LIN {X 0,Y 340.456,Z 505.145,A -85,B 0,C 180,E1 -14305.856,E2 -14305.856} C_VEL
LIN {X 0,Y 340.517,Z 502.884,A -85,B 0,C 180,E1 -14307.19,E2 -14307.19} C_VEL
LIN {X 0,Y 341.184,Z 502.798,A -85,B 0,C 180,E1 -14309.999,E2 -14309.999} C_VEL
LIN {X 0,Y 341.171,Z 502.802,A -85,B 0,C 180,E1 -14312.361,E2 -14312.361} C_VEL
LIN {X 0,Y 341.077,Z 502.809,A -85,B 0,C 180,E1 -14317.101,E2 -14317.101} C_VEL
LIN {X 0,Y 340.872,Z 502.837,A -85,B 0,C 180,E1 -14320.693,E2 -14320.693} C_VEL
LIN {X 0,Y 340.863,Z 502.841,A -85,B 0,C 180,E1 -14324.324,E2 -14324.324} C_VEL
LIN {X 0,Y 340.838,Z 502.842,A -85,B 0,C 180,E1 -14328.466,E2 -14328.466} C_VEL
LIN {X 0,Y 340.754,Z 502.851,A -85,B 0,C 180,E1 -14331.856,E2 -14331.856} C_VEL
LIN {X 0,Y 340.773,Z 502.848,A -85,B 0,C 180,E1 -14335.664,E2 -14335.664} C_VEL
LIN {X 0,Y 340.742,Z 502.855,A -85,B 0,C 180,E1 -14338.319,E2 -14338.319} C_VEL
LIN {X 0,Y 340.704,Z 502.855,A -85,B 0,C 180,E1 -14341.043,E2 -14341.043} C_VEL
LIN {X 0,Y 340.717,Z 502.854,A -85,B 0,C 180,E1 -14345.278,E2 -14345.278} C_VEL
LIN {X 0,Y 340.709,Z 502.858,A -85,B 0,C 180,E1 -14348.386,E2 -14348.386} C_VEL
LIN {X 0,Y 340.719,Z 502.859,A -85,B 0,C 180,E1 -14352.049,E2 -14352.049} C_VEL
LIN {X 0,Y 340.721,Z 502.854,A -85,B 0,C 180,E1 -14355.467,E2 -14355.467} C_VEL
LIN {X 0,Y 340.722,Z 502.853,A -85,B 0,C 180,E1 -14358.81,E2 -14358.81} C_VEL
LIN {X 0,Y 340.063,Z 502.939,A -85,B 0,C 180,E1 -14359.797,E2 -14359.797} C_VEL
LIN {X 0,Y 337.229,Z 503.295,A -85,B 0,C 180,E1 -14361.402,E2 -14361.402} C_VEL
LIN {X 0,Y 334.812,Z 503.598,A -85,B 0,C 180,E1 -14362.702,E2 -14362.702} C_VEL
LIN {X 0,Y 333.759,Z 503.725,A -85,B 0,C 180,E1 -14363.708,E2 -14363.708} C_VEL
LIN {X 0,Y 333.664,Z 503.734,A -85,B 0,C 180,E1 -14364.048,E2 -14364.048} C_VEL
LIN {X 0,Y 333.641,Z 503.736,A -85,B 0,C 180,E1 -14367.413,E2 -14367.413} C_VEL
LIN {X 0,Y 333.708,Z 503.726,A -85,B 0,C 180,E1 -14371.028,E2 -14371.028} C_VEL
LIN {X 0,Y 333.733,Z 503.727,A -85,B 0,C 180,E1 -14373.753,E2 -14373.753} C_VEL
LIN {X 0,Y 333.717,Z 503.731,A -85,B 0,C 180,E1 -14377.914,E2 -14377.914} C_VEL
LIN {X 0,Y 333.792,Z 503.719,A -85,B 0,C 180,E1 -14381.589,E2 -14381.589} C_VEL
LIN {X 0,Y 333.805,Z 503.717,A -85,B 0,C 180,E1 -14385.576,E2 -14385.576} C_VEL
LIN {X 0,Y 333.835,Z 503.711,A -85,B 0,C 180,E1 -14389.078,E2 -14389.078} C_VEL
LIN {X 0,Y 334.023,Z 503.687,A -85,B 0,C 180,E1 -14392.747,E2 -14392.747} C_VEL
LIN {X 0,Y 333.81,Z 503.714,A -85,B 0,C 180,E1 -14395.169,E2 -14395.169} C_VEL
LIN {X 0,Y 334.105,Z 503.681,A -85,B 0,C 180,E1 -14397.589,E2 -14397.589} C_VEL
LIN {X 0,Y 334.245,Z 503.663,A -85,B 0,C 180,E1 -14400,E2 -14400} C_VEL
LIN {X 0,Y 334.106,Z 503.678,A -85,B 0,C 180,E1 -14402.411,E2 -14402.411} C_VEL
LIN {X 0,Y 334.023,Z 503.689,A -85,B 0,C 180,E1 -14407.252,E2 -14407.252} C_VEL
LIN {X 0,Y 333.832,Z 503.711,A -85,B 0,C 180,E1 -14410.922,E2 -14410.922} C_VEL
LIN {X 0,Y 333.805,Z 503.714,A -85,B 0,C 180,E1 -14414.634,E2 -14414.634} C_VEL
LIN {X 0,Y 333.793,Z 503.716,A -85,B 0,C 180,E1 -14418.655,E2 -14418.655} C_VEL
LIN {X 0,Y 333.689,Z 503.73,A -85,B 0,C 180,E1 -14422.278,E2 -14422.278} C_VEL
LIN {X 0,Y 333.733,Z 503.724,A -85,B 0,C 180,E1 -14426.246,E2 -14426.246} C_VEL
LIN {X 0,Y 333.709,Z 503.727,A -85,B 0,C 180,E1 -14428.972,E2 -14428.972} C_VEL
LIN {X 0,Y 333.648,Z 503.734,A -85,B 0,C 180,E1 -14432.589,E2 -14432.589} C_VEL
LIN {X 0,Y 333.674,Z 503.732,A -85,B 0,C 180,E1 -14436.139,E2 -14436.139} C_VEL
LIN {X 0,Y 333.644,Z 503.737,A -85,B 0,C 180,E1 -14439.193,E2 -14439.193} C_VEL
LIN {X 0,Y 333.63,Z 503.736,A -85,B 0,C 180,E1 -14442.5,E2 -14442.5} C_VEL
LIN {X 0,Y 333.645,Z 503.736,A -85,B 0,C 180,E1 -14445.964,E2 -14445.964} C_VEL
LIN {X 0,Y 333.654,Z 503.738,A -85,B 0,C 180,E1 -14449.314,E2 -14449.314} C_VEL
LIN {X 0,Y 333.787,Z 503.868,A -85,B 0,C 180,E1 -14452.482,E2 -14452.482} C_VEL
LIN {X 0,Y 334.922,Z 510.332,A -85,B 0,C 180,E1 -14456.216,E2 -14456.216} C_VEL
LIN {X 0,Y 335.329,Z 513.013,A -85,B 0,C 180,E1 -14457.717,E2 -14457.717} C_VEL
LIN {X 0,Y 334.834,Z 518.114,A -85,B 0,C 180,E1 -14460.446,E2 -14460.446} C_VEL
LIN {X 0,Y 333.958,Z 525.622,A -85,B 0,C 180,E1 -14464.379,E2 -14464.379} C_VEL
LIN {X 0,Y 333.231,Z 532.887,A -85,B 0,C 180,E1 -14468.122,E2 -14468.122} C_VEL
LIN {X 0,Y 332.697,Z 540.288,A -85,B 0,C 180,E1 -14471.914,E2 -14471.914} C_VEL
LIN {X 0,Y 332.542,Z 543.414,A -85,B 0,C 180,E1 -14473.502,E2 -14473.502} C_VEL
LIN {X 0,Y 333.88,Z 554.918,A -85,B 0,C 180,E1 -14474.002,E2 -14474.002} C_VEL
LIN {X 0,Y 334.682,Z 563.382,A -85,B 0,C 180,E1 -14474.509,E2 -14474.509} C_VEL
LIN {X 0,Y 335.194,Z 571.374,A -85,B 0,C 180,E1 -14475.115,E2 -14475.115} C_VEL
LIN {X 0,Y 335.488,Z 578.299,A -85,B 0,C 180,E1 -14475.751,E2 -14475.751} C_VEL
LIN {X 0,Y 334.937,Z 586.572,A -85,B 0,C 180,E1 -14476.656,E2 -14476.656} C_VEL
LIN {X 0,Y 334.225,Z 594.387,A -85,B 0,C 180,E1 -14477.708,E2 -14477.708} C_VEL
LIN {X 0,Y 333.675,Z 600.834,A -85,B 0,C 180,E1 -14478.766,E2 -14478.766} C_VEL
LIN {X 0,Y 333.106,Z 606.952,A -85,B 0,C 180,E1 -14479.977,E2 -14479.977} C_VEL
LIN {X 0,Y 332.646,Z 613.19,A -85,B 0,C 180,E1 -14481.496,E2 -14481.496} C_VEL
LIN {X 0,Y 332.216,Z 618.901,A -85,B 0,C 180,E1 -14483.319,E2 -14483.319} C_VEL
LIN {X 0,Y 332.065,Z 621.825,A -85,B 0,C 180,E1 -14484.512,E2 -14484.512} C_VEL
LIN {X 0,Y 332.055,Z 625.07,A -85,B 0,C 180,E1 -14486.36,E2 -14486.36} C_VEL
LIN {X 0,Y 331.969,Z 626.568,A -85,B 0,C 180,E1 -14487.574,E2 -14487.574} C_VEL
LIN {X 0,Y 331.973,Z 627.512,A -85,B 0,C 180,E1 -14488.788,E2 -14488.788} C_VEL
LIN {X 0,Y 332.038,Z 627.871,A -85,B 0,C 180,E1 -14490.001,E2 -14490.001} C_VEL
LIN {X 0,Y 331.97,Z 627.733,A -85,B 0,C 180,E1 -14491.214,E2 -14491.214} C_VEL
LIN {X 0,Y 331.964,Z 627.113,A -85,B 0,C 180,E1 -14492.427,E2 -14492.427} C_VEL
LIN {X 0,Y 332.051,Z 626.001,A -85,B 0,C 180,E1 -14493.641,E2 -14493.641} C_VEL
LIN {X 0,Y 332.1,Z 624.338,A -85,B 0,C 180,E1 -14494.856,E2 -14494.856} C_VEL
LIN {X 0,Y 332.553,Z 618.216,A -85,B 0,C 180,E1 -14497.896,E2 -14497.896} C_VEL
LIN {X 0,Y 333.215,Z 613.214,A -85,B 0,C 180,E1 -14499.715,E2 -14499.715} C_VEL
LIN {X 0,Y 334.003,Z 607.935,A -85,B 0,C 180,E1 -14501.224,E2 -14501.224} C_VEL
LIN {X 0,Y 335.091,Z 601.437,A -85,B 0,C 180,E1 -14502.723,E2 -14502.723} C_VEL
LIN {X 0,Y 336.316,Z 593.514,A -85,B 0,C 180,E1 -14504.214,E2 -14504.214} C_VEL
LIN {X 0,Y 337.945,Z 583.56,A -85,B 0,C 180,E1 -14505.686,E2 -14505.686} C_VEL
LIN {X 0,Y 338.393,Z 575.402,A -85,B 0,C 180,E1 -14506.733,E2 -14506.733} C_VEL
LIN {X 0,Y 338.314,Z 568.475,A -85,B 0,C 180,E1 -14507.531,E2 -14507.531} C_VEL
LIN {X 0,Y 337.193,Z 558.94,A -85,B 0,C 180,E1 -14508.552,E2 -14508.552} C_VEL
LIN {X 0,Y 335.395,Z 550.189,A -85,B 0,C 180,E1 -14509.448,E2 -14509.448} C_VEL
LIN {X 0,Y 333.241,Z 542.09,A -85,B 0,C 180,E1 -14510.224,E2 -14510.224} C_VEL
LIN {X 0,Y 333.215,Z 541.572,A -85,B 0,C 180,E1 -14510.366,E2 -14510.366} C_VEL
LIN {X 0,Y 333.935,Z 535.173,A -85,B 0,C 180,E1 -14514.23,E2 -14514.23} C_VEL
LIN {X 0,Y 334.748,Z 530.134,A -85,B 0,C 180,E1 -14517.51,E2 -14517.51} C_VEL
LIN {X 0,Y 335.654,Z 525.473,A -85,B 0,C 180,E1 -14520.855,E2 -14520.855} C_VEL
LIN {X 0,Y 336.223,Z 522.467,A -85,B 0,C 180,E1 -14523.268,E2 -14523.268} C_VEL
LIN {X 0,Y 336.353,Z 519.746,A -85,B 0,C 180,E1 -14525.807,E2 -14525.807} C_VEL
LIN {X 0,Y 336.02,Z 517.109,A -85,B 0,C 180,E1 -14528.864,E2 -14528.864} C_VEL
LIN {X 0,Y 335.687,Z 514.987,A -85,B 0,C 180,E1 -14532.065,E2 -14532.065} C_VEL
LIN {X 0,Y 335.387,Z 513.454,A -85,B 0,C 180,E1 -14535.437,E2 -14535.437} C_VEL
LIN {X 0,Y 335.245,Z 512.57,A -85,B 0,C 180,E1 -14539,E2 -14539} C_VEL
LIN {X 0,Y 335.145,Z 512.414,A -85,B 0,C 180,E1 -14542.546,E2 -14542.546} C_VEL
LIN {X 0,Y 335.113,Z 512.774,A -85,B 0,C 180,E1 -14545.511,E2 -14545.511} C_VEL
LIN {X 0,Y 334.894,Z 513.56,A -85,B 0,C 180,E1 -14548.356,E2 -14548.356} C_VEL
LIN {X 0,Y 334.407,Z 515.069,A -85,B 0,C 180,E1 -14551.969,E2 -14551.969} C_VEL
LIN {X 0,Y 333.979,Z 516.753,A -85,B 0,C 180,E1 -14555.111,E2 -14555.111} C_VEL
LIN {X 0,Y 333.557,Z 519.216,A -85,B 0,C 180,E1 -14559.011,E2 -14559.011} C_VEL
LIN {X 0,Y 333.507,Z 520.041,A -85,B 0,C 180,E1 -14559.935,E2 -14559.935} C_VEL
LIN {X 0,Y 337.947,Z 531.73,A -85,B 0,C 180,E1 -14561.371,E2 -14561.371} C_VEL
LIN {X 0,Y 340.475,Z 541.669,A -85,B 0,C 180,E1 -14562.641,E2 -14562.641} C_VEL
LIN {X 0,Y 341.129,Z 546.298,A -85,B 0,C 180,E1 -14563.236,E2 -14563.236} C_VEL
LIN {X 0,Y 339.871,Z 554.77,A -85,B 0,C 180,E1 -14564.252,E2 -14564.252} C_VEL
LIN {X 0,Y 338.492,Z 563.651,A -85,B 0,C 180,E1 -14565.573,E2 -14565.573} C_VEL
LIN {X 0,Y 337.09,Z 571.617,A -85,B 0,C 180,E1 -14567.049,E2 -14567.049} C_VEL
LIN {X 0,Y 335.873,Z 577.991,A -85,B 0,C 180,E1 -14568.534,E2 -14568.534} C_VEL
LIN {X 0,Y 335.057,Z 582.231,A -85,B 0,C 180,E1 -14569.73,E2 -14569.73} C_VEL
LIN {X 0,Y 334.387,Z 586.055,A -85,B 0,C 180,E1 -14571.053,E2 -14571.053} C_VEL
LIN {X 0,Y 333.402,Z 589.807,A -85,B 0,C 180,E1 -14572.734,E2 -14572.734} C_VEL
LIN {X 0,Y 333.118,Z 591.829,A -85,B 0,C 180,E1 -14573.945,E2 -14573.945} C_VEL
LIN {X 0,Y 332.982,Z 593.306,A -85,B 0,C 180,E1 -14575.157,E2 -14575.157} C_VEL
LIN {X 0,Y 332.648,Z 594.219,A -85,B 0,C 180,E1 -14576.366,E2 -14576.366} C_VEL
LIN {X 0,Y 332.405,Z 594.638,A -85,B 0,C 180,E1 -14577.577,E2 -14577.577} C_VEL
LIN {X 0,Y 332.209,Z 594.58,A -85,B 0,C 180,E1 -14578.788,E2 -14578.788} C_VEL
LIN {X 0,Y 332.136,Z 594.037,A -85,B 0,C 180,E1 -14580,E2 -14580} C_VEL
LIN {X 0,Y 332.096,Z 592.929,A -85,B 0,C 180,E1 -14581.213,E2 -14581.213} C_VEL
LIN {X 0,Y 332.155,Z 590.254,A -85,B 0,C 180,E1 -14583.032,E2 -14583.032} C_VEL
LIN {X 0,Y 332.366,Z 586.242,A -85,B 0,C 180,E1 -14584.852,E2 -14584.852} C_VEL
LIN {X 0,Y 332.593,Z 580.732,A -85,B 0,C 180,E1 -14586.703,E2 -14586.703} C_VEL
LIN {X 0,Y 332.978,Z 575.054,A -85,B 0,C 180,E1 -14588.191,E2 -14588.191} C_VEL
LIN {X 0,Y 333.406,Z 567.758,A -85,B 0,C 180,E1 -14589.709,E2 -14589.709} C_VEL
LIN {X 0,Y 334.005,Z 559.596,A -85,B 0,C 180,E1 -14591.07,E2 -14591.07} C_VEL
LIN {X 0,Y 334.497,Z 551.909,A -85,B 0,C 180,E1 -14592.129,E2 -14592.129} C_VEL
LIN {X 0,Y 335.116,Z 542.576,A -85,B 0,C 180,E1 -14593.184,E2 -14593.184} C_VEL
LIN {X 0,Y 335.377,Z 535.383,A -85,B 0,C 180,E1 -14593.844,E2 -14593.844} C_VEL
LIN {X 0,Y 333.631,Z 524.142,A -85,B 0,C 180,E1 -14594.72,E2 -14594.72} C_VEL
LIN {X 0,Y 332.344,Z 514.848,A -85,B 0,C 180,E1 -14595.288,E2 -14595.288} C_VEL
LIN {X 0,Y 332.367,Z 511.054,A -85,B 0,C 180,E1 -14598.493,E2 -14598.493} C_VEL
LIN {X 0,Y 332.502,Z 506.577,A -85,B 0,C 180,E1 -14602.362,E2 -14602.362} C_VEL
LIN {X 0,Y 332.729,Z 503.94,A -85,B 0,C 180,E1 -14604.792,E2 -14604.792} C_VEL
LIN {X 0,Y 333.7,Z 507.775,A -85,B 0,C 180,E1 -14606.924,E2 -14606.924} C_VEL
LIN {X 0,Y 333.738,Z 511.614,A -85,B 0,C 180,E1 -14608.97,E2 -14608.97} C_VEL
LIN {X 0,Y 333.445,Z 518.337,A -85,B 0,C 180,E1 -14612.533,E2 -14612.533} C_VEL
LIN {X 0,Y 333.168,Z 525.241,A -85,B 0,C 180,E1 -14616.203,E2 -14616.203} C_VEL
LIN {X 0,Y 332.985,Z 529.458,A -85,B 0,C 180,E1 -14618.447,E2 -14618.447} C_VEL
LIN {X 0,Y 335.211,Z 539.502,A -85,B 0,C 180,E1 -14619.054,E2 -14619.054} C_VEL
LIN {X 0,Y 336.797,Z 548.312,A -85,B 0,C 180,E1 -14619.721,E2 -14619.721} C_VEL
LIN {X 0,Y 337.709,Z 557.401,A -85,B 0,C 180,E1 -14620.536,E2 -14620.536} C_VEL
LIN {X 0,Y 336.681,Z 568.368,A -85,B 0,C 180,E1 -14621.691,E2 -14621.691} C_VEL
LIN {X 0,Y 335.879,Z 575.943,A -85,B 0,C 180,E1 -14622.714,E2 -14622.714} C_VEL
LIN {X 0,Y 335.09,Z 582.589,A -85,B 0,C 180,E1 -14623.799,E2 -14623.799} C_VEL
LIN {X 0,Y 334.457,Z 587.63,A -85,B 0,C 180,E1 -14624.769,E2 -14624.769} C_VEL
LIN {X 0,Y 333.838,Z 592.947,A -85,B 0,C 180,E1 -14625.994,E2 -14625.994} C_VEL
LIN {X 0,Y 333.201,Z 598.466,A -85,B 0,C 180,E1 -14627.581,E2 -14627.581} C_VEL
LIN {X 0,Y 332.708,Z 602.588,A -85,B 0,C 180,E1 -14629.092,E2 -14629.092} C_VEL
LIN {X 0,Y 332.368,Z 605.767,A -85,B 0,C 180,E1 -14630.627,E2 -14630.627} C_VEL
LIN {X 0,Y 332.056,Z 608.005,A -85,B 0,C 180,E1 -14632.135,E2 -14632.135} C_VEL
LIN {X 0,Y 331.839,Z 609.408,A -85,B 0,C 180,E1 -14633.628,E2 -14633.628} C_VEL
LIN {X 0,Y 331.711,Z 610.143,A -85,B 0,C 180,E1 -14635.721,E2 -14635.721} C_VEL
LIN {X 0,Y 331.808,Z 609.081,A -85,B 0,C 180,E1 -14638.026,E2 -14638.026} C_VEL
LIN {X 0,Y 332.099,Z 606.537,A -85,B 0,C 180,E1 -14640.188,E2 -14640.188} C_VEL
LIN {X 0,Y 332.295,Z 603.919,A -85,B 0,C 180,E1 -14641.583,E2 -14641.583} C_VEL
LIN {X 0,Y 332.639,Z 600.056,A -85,B 0,C 180,E1 -14643.132,E2 -14643.132} C_VEL
LIN {X 0,Y 333.104,Z 594.919,A -85,B 0,C 180,E1 -14644.707,E2 -14644.707} C_VEL
LIN {X 0,Y 333.646,Z 589.34,A -85,B 0,C 180,E1 -14646.078,E2 -14646.078} C_VEL
LIN {X 0,Y 334.28,Z 582.643,A -85,B 0,C 180,E1 -14647.416,E2 -14647.416} C_VEL
LIN {X 0,Y 334.967,Z 575.255,A -85,B 0,C 180,E1 -14648.62,E2 -14648.62} C_VEL
LIN {X 0,Y 335.804,Z 565.471,A -85,B 0,C 180,E1 -14649.891,E2 -14649.891} C_VEL
LIN {X 0,Y 336.497,Z 556.393,A -85,B 0,C 180,E1 -14650.794,E2 -14650.794} C_VEL
LIN {X 0,Y 335.496,Z 547.321,A -85,B 0,C 180,E1 -14651.567,E2 -14651.567} C_VEL
LIN {X 0,Y 334.038,Z 537.768,A -85,B 0,C 180,E1 -14652.213,E2 -14652.213} C_VEL
LIN {X 0,Y 332.553,Z 529.31,A -85,B 0,C 180,E1 -14652.684,E2 -14652.684} C_VEL
LIN {X 0,Y 332.785,Z 522.475,A -85,B 0,C 180,E1 -14656.567,E2 -14656.567} C_VEL
LIN {X 0,Y 333.016,Z 515.913,A -85,B 0,C 180,E1 -14660.279,E2 -14660.279} C_VEL
LIN {X 0,Y 333.227,Z 510.519,A -85,B 0,C 180,E1 -14663.338,E2 -14663.338} C_VEL
LIN {X 0,Y 333.412,Z 506.235,A -85,B 0,C 180,E1 -14665.768,E2 -14665.768} C_VEL
LIN {X 0,Y 333.492,Z 503.758,A -85,B 0,C 180,E1 -14667.282,E2 -14667.282} C_VEL
LIN {X 0,Y 333.958,Z 503.697,A -85,B 0,C 180,E1 -14668.794,E2 -14668.794} C_VEL
LIN {X 0,Y 334.09,Z 503.679,A -85,B 0,C 180,E1 -14671.205,E2 -14671.205} C_VEL
LIN {X 0,Y 334.108,Z 503.682,A -85,B 0,C 180,E1 -14672.411,E2 -14672.411} C_VEL
LIN {X 0,Y 334.027,Z 503.687,A -85,B 0,C 180,E1 -14677.252,E2 -14677.252} C_VEL
LIN {X 0,Y 333.834,Z 503.711,A -85,B 0,C 180,E1 -14680.921,E2 -14680.921} C_VEL
LIN {X 0,Y 333.809,Z 503.716,A -85,B 0,C 180,E1 -14684.634,E2 -14684.634} C_VEL
LIN {X 0,Y 333.797,Z 503.717,A -85,B 0,C 180,E1 -14688.655,E2 -14688.655} C_VEL
LIN {X 0,Y 333.692,Z 503.734,A -85,B 0,C 180,E1 -14692.277,E2 -14692.277} C_VEL
LIN {X 0,Y 333.736,Z 503.728,A -85,B 0,C 180,E1 -14696.246,E2 -14696.246} C_VEL
LIN {X 0,Y 333.711,Z 503.726,A -85,B 0,C 180,E1 -14698.971,E2 -14698.971} C_VEL
LIN {X 0,Y 333.645,Z 503.736,A -85,B 0,C 180,E1 -14702.587,E2 -14702.587} C_VEL
LIN {X 0,Y 333.675,Z 503.736,A -85,B 0,C 180,E1 -14706.138,E2 -14706.138} C_VEL
LIN {X 0,Y 333.646,Z 503.734,A -85,B 0,C 180,E1 -14709.192,E2 -14709.192} C_VEL
LIN {X 0,Y 333.664,Z 503.734,A -85,B 0,C 180,E1 -14712.506,E2 -14712.506} C_VEL
LIN {X 0,Y 333.678,Z 503.735,A -85,B 0,C 180,E1 -14715.968,E2 -14715.968} C_VEL
LIN {X 0,Y 333.699,Z 503.728,A -85,B 0,C 180,E1 -14719.304,E2 -14719.304} C_VEL
LIN {X 0,Y 333.664,Z 503.732,A -85,B 0,C 180,E1 -14723.167,E2 -14723.167} C_VEL
LIN {X 0,Y 333.664,Z 503.734,A -85,B 0,C 180,E1 -14724.048,E2 -14724.048} C_VEL
LIN {X 0,Y 332.98,Z 503.818,A -85,B 0,C 180,E1 -14725.056,E2 -14725.056} C_VEL
LIN {X 0,Y 330.146,Z 504.171,A -85,B 0,C 180,E1 -14726.696,E2 -14726.696} C_VEL
LIN {X 0,Y 327.754,Z 504.473,A -85,B 0,C 180,E1 -14728.025,E2 -14728.025} C_VEL
LIN {X 0,Y 326.723,Z 504.599,A -85,B 0,C 180,E1 -14729.052,E2 -14729.052} C_VEL
LIN {X 0,Y 326.636,Z 504.608,A -85,B 0,C 180,E1 -14729.4,E2 -14729.4} C_VEL
LIN {X 0,Y 326.681,Z 504.602,A -85,B 0,C 180,E1 -14733.142,E2 -14733.142} C_VEL
LIN {X 0,Y 326.649,Z 504.611,A -85,B 0,C 180,E1 -14735.871,E2 -14735.871} C_VEL
LIN {X 0,Y 326.662,Z 504.609,A -85,B 0,C 180,E1 -14739.865,E2 -14739.865} C_VEL
LIN {X 0,Y 326.697,Z 504.601,A -85,B 0,C 180,E1 -14742.472,E2 -14742.472} C_VEL
LIN {X 0,Y 326.758,Z 504.594,A -85,B 0,C 180,E1 -14746.314,E2 -14746.314} C_VEL
LIN {X 0,Y 326.813,Z 504.588,A -85,B 0,C 180,E1 -14750.094,E2 -14750.094} C_VEL
LIN {X 0,Y 326.977,Z 504.565,A -85,B 0,C 180,E1 -14752.59,E2 -14752.59} C_VEL
LIN {X 0,Y 326.777,Z 504.59,A -85,B 0,C 180,E1 -14755.065,E2 -14755.065} C_VEL
LIN {X 0,Y 327.046,Z 504.559,A -85,B 0,C 180,E1 -14757.537,E2 -14757.537} C_VEL
LIN {X 0,Y 327.196,Z 504.541,A -85,B 0,C 180,E1 -14760,E2 -14760} C_VEL
LIN {X 0,Y 327.046,Z 504.557,A -85,B 0,C 180,E1 -14762.463,E2 -14762.463} C_VEL
LIN {X 0,Y 326.994,Z 504.564,A -85,B 0,C 180,E1 -14766.169,E2 -14766.169} C_VEL
LIN {X 0,Y 326.912,Z 504.573,A -85,B 0,C 180,E1 -14768.655,E2 -14768.655} C_VEL
LIN {X 0,Y 326.732,Z 504.596,A -85,B 0,C 180,E1 -14772.421,E2 -14772.421} C_VEL
LIN {X 0,Y 326.751,Z 504.593,A -85,B 0,C 180,E1 -14774.958,E2 -14774.958} C_VEL
LIN {X 0,Y 326.729,Z 504.596,A -85,B 0,C 180,E1 -14778.838,E2 -14778.838} C_VEL
LIN {X 0,Y 326.618,Z 504.609,A -85,B 0,C 180,E1 -14782.787,E2 -14782.787} C_VEL
LIN {X 0,Y 326.687,Z 504.605,A -85,B 0,C 180,E1 -14785.484,E2 -14785.484} C_VEL
LIN {X 0,Y 326.659,Z 504.609,A -85,B 0,C 180,E1 -14789.659,E2 -14789.659} C_VEL
LIN {X 0,Y 326.62,Z 504.61,A -85,B 0,C 180,E1 -14792.948,E2 -14792.948} C_VEL
LIN {X 0,Y 326.629,Z 504.61,A -85,B 0,C 180,E1 -14797.047,E2 -14797.047} C_VEL
LIN {X 0,Y 326.589,Z 504.614,A -85,B 0,C 180,E1 -14800.209,E2 -14800.209} C_VEL
LIN {X 0,Y 326.573,Z 504.621,A -85,B 0,C 180,E1 -14803.523,E2 -14803.523} C_VEL
LIN {X 0,Y 326.611,Z 504.612,A -85,B 0,C 180,E1 -14807.021,E2 -14807.021} C_VEL
LIN {X 0,Y 326.673,Z 504.608,A -85,B 0,C 180,E1 -14811.399,E2 -14811.399} C_VEL
LIN {X 0,Y 326.775,Z 504.712,A -85,B 0,C 180,E1 -14812.383,E2 -14812.383} C_VEL
LIN {X 0,Y 327.848,Z 511.059,A -85,B 0,C 180,E1 -14816.128,E2 -14816.128} C_VEL
LIN {X 0,Y 328.257,Z 513.695,A -85,B 0,C 180,E1 -14817.64,E2 -14817.64} C_VEL
LIN {X 0,Y 327.767,Z 518.822,A -85,B 0,C 180,E1 -14820.452,E2 -14820.452} C_VEL
LIN {X 0,Y 326.848,Z 526.428,A -85,B 0,C 180,E1 -14824.53,E2 -14824.53} C_VEL
LIN {X 0,Y 326.065,Z 533.957,A -85,B 0,C 180,E1 -14828.506,E2 -14828.506} C_VEL
LIN {X 0,Y 325.548,Z 541.393,A -85,B 0,C 180,E1 -14832.409,E2 -14832.409} C_VEL
LIN {X 0,Y 325.488,Z 542.866,A -85,B 0,C 180,E1 -14833.174,E2 -14833.174} C_VEL
LIN {X 0,Y 326.898,Z 554.924,A -85,B 0,C 180,E1 -14833.711,E2 -14833.711} C_VEL
LIN {X 0,Y 327.647,Z 563.055,A -85,B 0,C 180,E1 -14834.208,E2 -14834.208} C_VEL
LIN {X 0,Y 328.231,Z 571.872,A -85,B 0,C 180,E1 -14834.898,E2 -14834.898} C_VEL
LIN {X 0,Y 328.494,Z 579.168,A -85,B 0,C 180,E1 -14835.599,E2 -14835.599} C_VEL
LIN {X 0,Y 327.907,Z 587.253,A -85,B 0,C 180,E1 -14836.522,E2 -14836.522} C_VEL
LIN {X 0,Y 327.167,Z 594.921,A -85,B 0,C 180,E1 -14837.596,E2 -14837.596} C_VEL
LIN {X 0,Y 326.383,Z 603.72,A -85,B 0,C 180,E1 -14839.14,E2 -14839.14} C_VEL
LIN {X 0,Y 325.793,Z 610.485,A -85,B 0,C 180,E1 -14840.69,E2 -14840.69} C_VEL
LIN {X 0,Y 325.437,Z 614.926,A -85,B 0,C 180,E1 -14841.931,E2 -14841.931} C_VEL
LIN {X 0,Y 325.054,Z 620.12,A -85,B 0,C 180,E1 -14843.795,E2 -14843.795} C_VEL
LIN {X 0,Y 324.975,Z 623.913,A -85,B 0,C 180,E1 -14845.66,E2 -14845.66} C_VEL
LIN {X 0,Y 324.887,Z 626.343,A -85,B 0,C 180,E1 -14847.521,E2 -14847.521} C_VEL
LIN {X 0,Y 324.879,Z 627.292,A -85,B 0,C 180,E1 -14848.761,E2 -14848.761} C_VEL
LIN {X 0,Y 324.94,Z 627.668,A -85,B 0,C 180,E1 -14850.001,E2 -14850.001} C_VEL
LIN {X 0,Y 324.876,Z 627.552,A -85,B 0,C 180,E1 -14851.24,E2 -14851.24} C_VEL
LIN {X 0,Y 324.882,Z 626.955,A -85,B 0,C 180,E1 -14852.48,E2 -14852.48} C_VEL
LIN {X 0,Y 324.957,Z 625.869,A -85,B 0,C 180,E1 -14853.721,E2 -14853.721} C_VEL
LIN {X 0,Y 325.002,Z 624.215,A -85,B 0,C 180,E1 -14854.963,E2 -14854.963} C_VEL
LIN {X 0,Y 325.514,Z 618.279,A -85,B 0,C 180,E1 -14858.068,E2 -14858.068} C_VEL
LIN {X 0,Y 326.242,Z 613.522,A -85,B 0,C 180,E1 -14859.924,E2 -14859.924} C_VEL
LIN {X 0,Y 327.069,Z 608.384,A -85,B 0,C 180,E1 -14861.465,E2 -14861.465} C_VEL
LIN {X 0,Y 328.207,Z 602.073,A -85,B 0,C 180,E1 -14862.994,E2 -14862.994} C_VEL
LIN {X 0,Y 329.506,Z 594.438,A -85,B 0,C 180,E1 -14864.514,E2 -14864.514} C_VEL
LIN {X 0,Y 331.25,Z 585.018,A -85,B 0,C 180,E1 -14866.011,E2 -14866.011} C_VEL
LIN {X 0,Y 331.881,Z 575.754,A -85,B 0,C 180,E1 -14867.246,E2 -14867.246} C_VEL
LIN {X 0,Y 331.661,Z 567.872,A -85,B 0,C 180,E1 -14868.214,E2 -14868.214} C_VEL
LIN {X 0,Y 330.433,Z 557.952,A -85,B 0,C 180,E1 -14869.339,E2 -14869.339} C_VEL
LIN {X 0,Y 327.373,Z 545.084,A -85,B 0,C 180,E1 -14870.746,E2 -14870.746} C_VEL
LIN {X 0,Y 326.338,Z 541.196,A -85,B 0,C 180,E1 -14871.145,E2 -14871.145} C_VEL
LIN {X 0,Y 327.275,Z 534.181,A -85,B 0,C 180,E1 -14875.589,E2 -14875.589} C_VEL
LIN {X 0,Y 328.27,Z 528.603,A -85,B 0,C 180,E1 -14879.5,E2 -14879.5} C_VEL
LIN {X 0,Y 329.012,Z 525.066,A -85,B 0,C 180,E1 -14882.278,E2 -14882.278} C_VEL
LIN {X 0,Y 329.297,Z 523.413,A -85,B 0,C 180,E1 -14883.705,E2 -14883.705} C_VEL
LIN {X 0,Y 329.434,Z 521.217,A -85,B 0,C 180,E1 -14885.838,E2 -14885.838} C_VEL
LIN {X 0,Y 329.153,Z 519.145,A -85,B 0,C 180,E1 -14888.259,E2 -14888.259} C_VEL
LIN {X 0,Y 328.823,Z 516.872,A -85,B 0,C 180,E1 -14891.577,E2 -14891.577} C_VEL
LIN {X 0,Y 328.505,Z 515.196,A -85,B 0,C 180,E1 -14895.09,E2 -14895.09} C_VEL
LIN {X 0,Y 328.33,Z 514.25,A -85,B 0,C 180,E1 -14898.521,E2 -14898.521} C_VEL
LIN {X 0,Y 328.233,Z 513.962,A -85,B 0,C 180,E1 -14902.395,E2 -14902.395} C_VEL
LIN {X 0,Y 328.21,Z 514.155,A -85,B 0,C 180,E1 -14904.679,E2 -14904.679} C_VEL
LIN {X 0,Y 328.007,Z 514.789,A -85,B 0,C 180,E1 -14907.611,E2 -14907.611} C_VEL
LIN {X 0,Y 327.64,Z 515.787,A -85,B 0,C 180,E1 -14910.439,E2 -14910.439} C_VEL
LIN {X 0,Y 327.228,Z 517.05,A -85,B 0,C 180,E1 -14913.191,E2 -14913.191} C_VEL
LIN {X 0,Y 326.727,Z 519.3,A -85,B 0,C 180,E1 -14917.221,E2 -14917.221} C_VEL
LIN {X 0,Y 326.584,Z 520.565,A -85,B 0,C 180,E1 -14919.058,E2 -14919.058} C_VEL
LIN {X 0,Y 327.057,Z 522.242,A -85,B 0,C 180,E1 -14919.234,E2 -14919.234} C_VEL
LIN {X 0,Y 330.875,Z 531.6,A -85,B 0,C 180,E1 -14920.526,E2 -14920.526} C_VEL
LIN {X 0,Y 333.26,Z 539.691,A -85,B 0,C 180,E1 -14921.622,E2 -14921.622} C_VEL
LIN {X 0,Y 334.592,Z 546.372,A -85,B 0,C 180,E1 -14922.556,E2 -14922.556} C_VEL
LIN {X 0,Y 334.41,Z 550.188,A -85,B 0,C 180,E1 -14923.046,E2 -14923.046} C_VEL
LIN {X 0,Y 332.785,Z 560.085,A -85,B 0,C 180,E1 -14924.38,E2 -14924.38} C_VEL
LIN {X 0,Y 331.488,Z 567.188,A -85,B 0,C 180,E1 -14925.575,E2 -14925.575} C_VEL
LIN {X 0,Y 330.343,Z 573.146,A -85,B 0,C 180,E1 -14926.779,E2 -14926.779} C_VEL
LIN {X 0,Y 329.042,Z 579.275,A -85,B 0,C 180,E1 -14928.293,E2 -14928.293} C_VEL
LIN {X 0,Y 328.157,Z 583.323,A -85,B 0,C 180,E1 -14929.511,E2 -14929.511} C_VEL
LIN {X 0,Y 327.188,Z 588.154,A -85,B 0,C 180,E1 -14931.352,E2 -14931.352} C_VEL
LIN {X 0,Y 326.411,Z 590.63,A -85,B 0,C 180,E1 -14932.578,E2 -14932.578} C_VEL
LIN {X 0,Y 326.088,Z 592.528,A -85,B 0,C 180,E1 -14933.814,E2 -14933.814} C_VEL
LIN {X 0,Y 325.934,Z 593.923,A -85,B 0,C 180,E1 -14935.052,E2 -14935.052} C_VEL
LIN {X 0,Y 325.597,Z 594.77,A -85,B 0,C 180,E1 -14936.287,E2 -14936.287} C_VEL
LIN {X 0,Y 325.324,Z 595.07,A -85,B 0,C 180,E1 -14937.524,E2 -14937.524} C_VEL
LIN {X 0,Y 325.119,Z 594.898,A -85,B 0,C 180,E1 -14938.761,E2 -14938.761} C_VEL
LIN {X 0,Y 325.039,Z 594.245,A -85,B 0,C 180,E1 -14940,E2 -14940} C_VEL
LIN {X 0,Y 324.998,Z 593.085,A -85,B 0,C 180,E1 -14941.239,E2 -14941.239} C_VEL
LIN {X 0,Y 325.076,Z 590.216,A -85,B 0,C 180,E1 -14943.098,E2 -14943.098} C_VEL
LIN {X 0,Y 325.237,Z 587.663,A -85,B 0,C 180,E1 -14944.338,E2 -14944.338} C_VEL
LIN {X 0,Y 325.334,Z 584.452,A -85,B 0,C 180,E1 -14945.579,E2 -14945.579} C_VEL
LIN {X 0,Y 325.726,Z 578.244,A -85,B 0,C 180,E1 -14947.438,E2 -14947.438} C_VEL
LIN {X 0,Y 325.969,Z 573.133,A -85,B 0,C 180,E1 -14948.68,E2 -14948.68} C_VEL
LIN {X 0,Y 326.397,Z 567.037,A -85,B 0,C 180,E1 -14949.919,E2 -14949.919} C_VEL
LIN {X 0,Y 326.958,Z 558.716,A -85,B 0,C 180,E1 -14951.312,E2 -14951.312} C_VEL
LIN {X 0,Y 327.56,Z 549.627,A -85,B 0,C 180,E1 -14952.547,E2 -14952.547} C_VEL
LIN {X 0,Y 328.248,Z 539.472,A -85,B 0,C 180,E1 -14953.622,E2 -14953.622} C_VEL
LIN {X 0,Y 328.286,Z 535.898,A -85,B 0,C 180,E1 -14953.947,E2 -14953.947} C_VEL
LIN {X 0,Y 326.398,Z 523.837,A -85,B 0,C 180,E1 -14954.901,E2 -14954.901} C_VEL
LIN {X 0,Y 325.271,Z 515.176,A -85,B 0,C 180,E1 -14955.428,E2 -14955.428} C_VEL
LIN {X 0,Y 325.291,Z 511.118,A -85,B 0,C 180,E1 -14958.91,E2 -14958.91} C_VEL
LIN {X 0,Y 325.439,Z 507.836,A -85,B 0,C 180,E1 -14961.78,E2 -14961.78} C_VEL
LIN {X 0,Y 325.628,Z 504.921,A -85,B 0,C 180,E1 -14964.543,E2 -14964.543} C_VEL
LIN {X 0,Y 326.722,Z 508.987,A -85,B 0,C 180,E1 -14966.854,E2 -14966.854} C_VEL
LIN {X 0,Y 326.759,Z 512.81,A -85,B 0,C 180,E1 -14968.943,E2 -14968.943} C_VEL
LIN {X 0,Y 326.404,Z 520.155,A -85,B 0,C 180,E1 -14972.887,E2 -14972.887} C_VEL
LIN {X 0,Y 326.145,Z 526.532,A -85,B 0,C 180,E1 -14976.334,E2 -14976.334} C_VEL
LIN {X 0,Y 326.022,Z 529.782,A -85,B 0,C 180,E1 -14978.004,E2 -14978.004} C_VEL
LIN {X 0,Y 328.328,Z 539.758,A -85,B 0,C 180,E1 -14978.629,E2 -14978.629} C_VEL
LIN {X 0,Y 330.124,Z 550.005,A -85,B 0,C 180,E1 -14979.435,E2 -14979.435} C_VEL
LIN {X 0,Y 330.866,Z 558.92,A -85,B 0,C 180,E1 -14980.277,E2 -14980.277} C_VEL
LIN {X 0,Y 329.81,Z 569.292,A -85,B 0,C 180,E1 -14981.433,E2 -14981.433} C_VEL
LIN {X 0,Y 328.94,Z 576.979,A -85,B 0,C 180,E1 -14982.514,E2 -14982.514} C_VEL
LIN {X 0,Y 327.953,Z 584.959,A -85,B 0,C 180,E1 -14983.897,E2 -14983.897} C_VEL
LIN {X 0,Y 327.049,Z 592.194,A -85,B 0,C 180,E1 -14985.477,E2 -14985.477} C_VEL
LIN {X 0,Y 326.297,Z 597.855,A -85,B 0,C 180,E1 -14987.081,E2 -14987.081} C_VEL
LIN {X 0,Y 325.787,Z 602.098,A -85,B 0,C 180,E1 -14988.606,E2 -14988.606} C_VEL
LIN {X 0,Y 325.48,Z 604.453,A -85,B 0,C 180,E1 -14989.625,E2 -14989.625} C_VEL
LIN {X 0,Y 325.137,Z 607.162,A -85,B 0,C 180,E1 -14991.181,E2 -14991.181} C_VEL
LIN {X 0,Y 324.799,Z 609.349,A -85,B 0,C 180,E1 -14993.188,E2 -14993.188} C_VEL
LIN {X 0,Y 324.703,Z 610.038,A -85,B 0,C 180,E1 -14994.239,E2 -14994.239} C_VEL
LIN {X 0,Y 324.635,Z 610.324,A -85,B 0,C 180,E1 -14995.745,E2 -14995.745} C_VEL
LIN {X 0,Y 324.68,Z 609.612,A -85,B 0,C 180,E1 -14997.586,E2 -14997.586} C_VEL
LIN {X 0,Y 324.767,Z 608.707,A -85,B 0,C 180,E1 -14998.71,E2 -14998.71} C_VEL
LIN {X 0,Y 324.992,Z 606.811,A -85,B 0,C 180,E1 -15000.173,E2 -15000.173} C_VEL
LIN {X 0,Y 325.222,Z 604.188,A -85,B 0,C 180,E1 -15001.613,E2 -15001.613} C_VEL
LIN {X 0,Y 325.602,Z 599.769,A -85,B 0,C 180,E1 -15003.392,E2 -15003.392} C_VEL
LIN {X 0,Y 326.064,Z 595.041,A -85,B 0,C 180,E1 -15004.86,E2 -15004.86} C_VEL
LIN {X 0,Y 326.601,Z 589.701,A -85,B 0,C 180,E1 -15006.204,E2 -15006.204} C_VEL
LIN {X 0,Y 327.197,Z 583.63,A -85,B 0,C 180,E1 -15007.461,E2 -15007.461} C_VEL
LIN {X 0,Y 327.84,Z 576.806,A -85,B 0,C 180,E1 -15008.627,E2 -15008.627} C_VEL
LIN {X 0,Y 328.565,Z 569.456,A -85,B 0,C 180,E1 -15009.66,E2 -15009.66} C_VEL
LIN {X 0,Y 329.26,Z 560.558,A -85,B 0,C 180,E1 -15010.679,E2 -15010.679} C_VEL
LIN {X 0,Y 329.44,Z 555.314,A -85,B 0,C 180,E1 -15011.175,E2 -15011.175} C_VEL
LIN {X 0,Y 328.342,Z 546.652,A -85,B 0,C 180,E1 -15011.918,E2 -15011.918} C_VEL
LIN {X 0,Y 326.773,Z 536.63,A -85,B 0,C 180,E1 -15012.597,E2 -15012.597} C_VEL
LIN {X 0,Y 325.509,Z 529.501,A -85,B 0,C 180,E1 -15012.972,E2 -15012.972} C_VEL
LIN {X 0,Y 325.751,Z 522.645,A -85,B 0,C 180,E1 -15016.906,E2 -15016.906} C_VEL
LIN {X 0,Y 326.009,Z 515.996,A -85,B 0,C 180,E1 -15020.695,E2 -15020.695} C_VEL
LIN {X 0,Y 326.275,Z 509.457,A -85,B 0,C 180,E1 -15024.437,E2 -15024.437} C_VEL
LIN {X 0,Y 326.491,Z 504.63,A -85,B 0,C 180,E1 -15027.378,E2 -15027.378} C_VEL
LIN {X 0,Y 327.092,Z 504.553,A -85,B 0,C 180,E1 -15029.999,E2 -15029.999} C_VEL
LIN {X 0,Y 327.049,Z 504.56,A -85,B 0,C 180,E1 -15032.463,E2 -15032.463} C_VEL
LIN {X 0,Y 326.998,Z 504.566,A -85,B 0,C 180,E1 -15036.168,E2 -15036.168} C_VEL
LIN {X 0,Y 326.916,Z 504.575,A -85,B 0,C 180,E1 -15038.654,E2 -15038.654} C_VEL
LIN {X 0,Y 326.736,Z 504.599,A -85,B 0,C 180,E1 -15042.421,E2 -15042.421} C_VEL
LIN {X 0,Y 326.755,Z 504.593,A -85,B 0,C 180,E1 -15044.957,E2 -15044.957} C_VEL
LIN {X 0,Y 326.734,Z 504.596,A -85,B 0,C 180,E1 -15048.838,E2 -15048.838} C_VEL
LIN {X 0,Y 326.621,Z 504.61,A -85,B 0,C 180,E1 -15052.787,E2 -15052.787} C_VEL
LIN {X 0,Y 326.69,Z 504.601,A -85,B 0,C 180,E1 -15055.483,E2 -15055.483} C_VEL
LIN {X 0,Y 326.672,Z 504.608,A -85,B 0,C 180,E1 -15058.248,E2 -15058.248} C_VEL
LIN {X 0,Y 326.594,Z 504.612,A -85,B 0,C 180,E1 -15061.094,E2 -15061.094} C_VEL
LIN {X 0,Y 326.607,Z 504.615,A -85,B 0,C 180,E1 -15064.019,E2 -15064.019} C_VEL
LIN {X 0,Y 326.627,Z 504.608,A -85,B 0,C 180,E1 -15067.238,E2 -15067.238} C_VEL
LIN {X 0,Y 326.583,Z 504.614,A -85,B 0,C 180,E1 -15071.132,E2 -15071.132} C_VEL
LIN {X 0,Y 326.595,Z 504.613,A -85,B 0,C 180,E1 -15074.755,E2 -15074.755} C_VEL
LIN {X 0,Y 326.621,Z 504.614,A -85,B 0,C 180,E1 -15078.161,E2 -15078.161} C_VEL
LIN {X 0,Y 326.645,Z 504.607,A -85,B 0,C 180,E1 -15081.394,E2 -15081.394} C_VEL
LIN {X 0,Y 326.617,Z 504.61,A -85,B 0,C 180,E1 -15084.851,E2 -15084.851} C_VEL
LIN {X 0,Y 326.605,Z 504.612,A -85,B 0,C 180,E1 -15087.455,E2 -15087.455} C_VEL
LIN {X 0,Y 326.636,Z 504.608,A -85,B 0,C 180,E1 -15089.4,E2 -15089.4} C_VEL
LIN {X 0,Y 325.965,Z 504.693,A -85,B 0,C 180,E1 -15090.429,E2 -15090.429} C_VEL
LIN {X 0,Y 323.133,Z 505.048,A -85,B 0,C 180,E1 -15092.104,E2 -15092.104} C_VEL
LIN {X 0,Y 320.733,Z 505.345,A -85,B 0,C 180,E1 -15093.461,E2 -15093.461} C_VEL
LIN {X 0,Y 319.694,Z 505.473,A -85,B 0,C 180,E1 -15094.511,E2 -15094.511} C_VEL
LIN {X 0,Y 319.605,Z 505.483,A -85,B 0,C 180,E1 -15094.866,E2 -15094.866} C_VEL
LIN {X 0,Y 319.594,Z 505.489,A -85,B 0,C 180,E1 -15098.047,E2 -15098.047} C_VEL
LIN {X 0,Y 319.687,Z 505.473,A -85,B 0,C 180,E1 -15100.962,E2 -15100.962} C_VEL
LIN {X 0,Y 319.728,Z 505.469,A -85,B 0,C 180,E1 -15105.275,E2 -15105.275} C_VEL
LIN {X 0,Y 319.757,Z 505.47,A -85,B 0,C 180,E1 -15109.873,E2 -15109.873} C_VEL
LIN {X 0,Y 319.931,Z 505.443,A -85,B 0,C 180,E1 -15112.426,E2 -15112.426} C_VEL
LIN {X 0,Y 319.746,Z 505.465,A -85,B 0,C 180,E1 -15114.956,E2 -15114.956} C_VEL
LIN {X 0,Y 319.99,Z 505.438,A -85,B 0,C 180,E1 -15117.482,E2 -15117.482} C_VEL
LIN {X 0,Y 320.148,Z 505.419,A -85,B 0,C 180,E1 -15120,E2 -15120} C_VEL
LIN {X 0,Y 319.99,Z 505.435,A -85,B 0,C 180,E1 -15122.518,E2 -15122.518} C_VEL
LIN {X 0,Y 319.95,Z 505.441,A -85,B 0,C 180,E1 -15126.305,E2 -15126.305} C_VEL
LIN {X 0,Y 319.84,Z 505.454,A -85,B 0,C 180,E1 -15128.848,E2 -15128.848} C_VEL
LIN {X 0,Y 319.679,Z 505.474,A -85,B 0,C 180,E1 -15132.7,E2 -15132.7} C_VEL
LIN {X 0,Y 319.696,Z 505.474,A -85,B 0,C 180,E1 -15135.296,E2 -15135.296} C_VEL
LIN {X 0,Y 319.671,Z 505.477,A -85,B 0,C 180,E1 -15139.255,E2 -15139.255} C_VEL
LIN {X 0,Y 319.567,Z 505.491,A -85,B 0,C 180,E1 -15143.32,E2 -15143.32} C_VEL
LIN {X 0,Y 319.632,Z 505.481,A -85,B 0,C 180,E1 -15146.088,E2 -15146.088} C_VEL
LIN {X 0,Y 319.587,Z 505.486,A -85,B 0,C 180,E1 -15148.934,E2 -15148.934} C_VEL
LIN {X 0,Y 319.536,Z 505.495,A -85,B 0,C 180,E1 -15151.861,E2 -15151.861} C_VEL
LIN {X 0,Y 319.578,Z 505.492,A -85,B 0,C 180,E1 -15155.544,E2 -15155.544} C_VEL
LIN {X 0,Y 319.571,Z 505.489,A -85,B 0,C 180,E1 -15158.008,E2 -15158.008} C_VEL
LIN {X 0,Y 319.549,Z 505.495,A -85,B 0,C 180,E1 -15161.603,E2 -15161.603} C_VEL
LIN {X 0,Y 319.549,Z 505.494,A -85,B 0,C 180,E1 -15165.269,E2 -15165.269} C_VEL
LIN {X 0,Y 319.544,Z 505.491,A -85,B 0,C 180,E1 -15168.715,E2 -15168.715} C_VEL
LIN {X 0,Y 319.726,Z 505.597,A -85,B 0,C 180,E1 -15172.309,E2 -15172.309} C_VEL
LIN {X 0,Y 320.88,Z 512.26,A -85,B 0,C 180,E1 -15176.334,E2 -15176.334} C_VEL
LIN {X 0,Y 321.184,Z 515.691,A -85,B 0,C 180,E1 -15178.322,E2 -15178.322} C_VEL
LIN {X 0,Y 320.325,Z 522.178,A -85,B 0,C 180,E1 -15181.929,E2 -15181.929} C_VEL
LIN {X 0,Y 319.462,Z 529.584,A -85,B 0,C 180,E1 -15185.985,E2 -15185.985} C_VEL
LIN {X 0,Y 318.768,Z 537.049,A -85,B 0,C 180,E1 -15190.018,E2 -15190.018} C_VEL
LIN {X 0,Y 318.422,Z 542.258,A -85,B 0,C 180,E1 -15192.831,E2 -15192.831} C_VEL
LIN {X 0,Y 319.859,Z 554.424,A -85,B 0,C 180,E1 -15193.383,E2 -15193.383} C_VEL
LIN {X 0,Y 320.702,Z 563.738,A -85,B 0,C 180,E1 -15193.973,E2 -15193.973} C_VEL
LIN {X 0,Y 321.313,Z 573.542,A -85,B 0,C 180,E1 -15194.784,E2 -15194.784} C_VEL
LIN {X 0,Y 321.412,Z 581.43,A -85,B 0,C 180,E1 -15195.599,E2 -15195.599} C_VEL
LIN {X 0,Y 320.509,Z 591.332,A -85,B 0,C 180,E1 -15196.851,E2 -15196.851} C_VEL
LIN {X 0,Y 319.878,Z 598.22,A -85,B 0,C 180,E1 -15197.953,E2 -15197.953} C_VEL
LIN {X 0,Y 319.242,Z 604.709,A -85,B 0,C 180,E1 -15199.216,E2 -15199.216} C_VEL
LIN {X 0,Y 318.756,Z 610.092,A -85,B 0,C 180,E1 -15200.482,E2 -15200.482} C_VEL
LIN {X 0,Y 318.388,Z 614.571,A -85,B 0,C 180,E1 -15201.751,E2 -15201.751} C_VEL
LIN {X 0,Y 318.1,Z 618.281,A -85,B 0,C 180,E1 -15203.021,E2 -15203.021} C_VEL
LIN {X 0,Y 317.884,Z 622.471,A -85,B 0,C 180,E1 -15204.927,E2 -15204.927} C_VEL
LIN {X 0,Y 317.889,Z 624.562,A -85,B 0,C 180,E1 -15206.198,E2 -15206.198} C_VEL
LIN {X 0,Y 317.808,Z 626.106,A -85,B 0,C 180,E1 -15207.466,E2 -15207.466} C_VEL
LIN {X 0,Y 317.789,Z 627.062,A -85,B 0,C 180,E1 -15208.733,E2 -15208.733} C_VEL
LIN {X 0,Y 317.844,Z 627.462,A -85,B 0,C 180,E1 -15210.001,E2 -15210.001} C_VEL
LIN {X 0,Y 317.786,Z 627.374,A -85,B 0,C 180,E1 -15211.268,E2 -15211.268} C_VEL
LIN {X 0,Y 317.803,Z 626.804,A -85,B 0,C 180,E1 -15212.536,E2 -15212.536} C_VEL
LIN {X 0,Y 317.866,Z 625.742,A -85,B 0,C 180,E1 -15213.804,E2 -15213.804} C_VEL
LIN {X 0,Y 317.916,Z 624.095,A -85,B 0,C 180,E1 -15215.074,E2 -15215.074} C_VEL
LIN {X 0,Y 318.475,Z 618.325,A -85,B 0,C 180,E1 -15218.248,E2 -15218.248} C_VEL
LIN {X 0,Y 319.245,Z 613.79,A -85,B 0,C 180,E1 -15220.144,E2 -15220.144} C_VEL
LIN {X 0,Y 320.395,Z 607.735,A -85,B 0,C 180,E1 -15222.028,E2 -15222.028} C_VEL
LIN {X 0,Y 321.623,Z 601.427,A -85,B 0,C 180,E1 -15223.587,E2 -15223.587} C_VEL
LIN {X 0,Y 322.712,Z 595.395,A -85,B 0,C 180,E1 -15224.827,E2 -15224.827} C_VEL
LIN {X 0,Y 324.163,Z 588.243,A -85,B 0,C 180,E1 -15226.048,E2 -15226.048} C_VEL
LIN {X 0,Y 325.172,Z 580.26,A -85,B 0,C 180,E1 -15227.243,E2 -15227.243} C_VEL
LIN {X 0,Y 325.379,Z 571.406,A -85,B 0,C 180,E1 -15228.431,E2 -15228.431} C_VEL
LIN {X 0,Y 324.397,Z 561.029,A -85,B 0,C 180,E1 -15229.714,E2 -15229.714} C_VEL
LIN {X 0,Y 322.29,Z 551.036,A -85,B 0,C 180,E1 -15230.904,E2 -15230.904} C_VEL
LIN {X 0,Y 319.901,Z 542.899,A -85,B 0,C 180,E1 -15231.86,E2 -15231.86} C_VEL
LIN {X 0,Y 319.456,Z 540.628,A -85,B 0,C 180,E1 -15232.111,E2 -15232.111} C_VEL
LIN {X 0,Y 320.349,Z 534.703,A -85,B 0,C 180,E1 -15236.026,E2 -15236.026} C_VEL
LIN {X 0,Y 321.13,Z 530.695,A -85,B 0,C 180,E1 -15238.907,E2 -15238.907} C_VEL
LIN {X 0,Y 321.855,Z 527.261,A -85,B 0,C 180,E1 -15241.614,E2 -15241.614} C_VEL
LIN {X 0,Y 322.39,Z 524.007,A -85,B 0,C 180,E1 -15244.528,E2 -15244.528} C_VEL
LIN {X 0,Y 322.44,Z 522.354,A -85,B 0,C 180,E1 -15246.248,E2 -15246.248} C_VEL
LIN {X 0,Y 322.102,Z 519.966,A -85,B 0,C 180,E1 -15249.255,E2 -15249.255} C_VEL
LIN {X 0,Y 321.794,Z 517.91,A -85,B 0,C 180,E1 -15252.614,E2 -15252.614} C_VEL
LIN {X 0,Y 321.518,Z 516.452,A -85,B 0,C 180,E1 -15256.166,E2 -15256.166} C_VEL
LIN {X 0,Y 321.356,Z 515.659,A -85,B 0,C 180,E1 -15259.947,E2 -15259.947} C_VEL
LIN {X 0,Y 321.32,Z 515.533,A -85,B 0,C 180,E1 -15262.235,E2 -15262.235} C_VEL
LIN {X 0,Y 321.211,Z 515.944,A -85,B 0,C 180,E1 -15266.247,E2 -15266.247} C_VEL
LIN {X 0,Y 320.777,Z 516.96,A -85,B 0,C 180,E1 -15269.741,E2 -15269.741} C_VEL
LIN {X 0,Y 320.347,Z 518.12,A -85,B 0,C 180,E1 -15272.567,E2 -15272.567} C_VEL
LIN {X 0,Y 319.792,Z 520.281,A -85,B 0,C 180,E1 -15276.698,E2 -15276.698} C_VEL
LIN {X 0,Y 319.646,Z 521.094,A -85,B 0,C 180,E1 -15278.081,E2 -15278.081} C_VEL
LIN {X 0,Y 320.277,Z 523.174,A -85,B 0,C 180,E1 -15278.331,E2 -15278.331} C_VEL
LIN {X 0,Y 323.095,Z 529.298,A -85,B 0,C 180,E1 -15279.285,E2 -15279.285} C_VEL
LIN {X 0,Y 326.262,Z 538.574,A -85,B 0,C 180,E1 -15280.638,E2 -15280.638} C_VEL
LIN {X 0,Y 328.215,Z 547.876,A -85,B 0,C 180,E1 -15282.03,E2 -15282.03} C_VEL
LIN {X 0,Y 328.262,Z 550.72,A -85,B 0,C 180,E1 -15282.427,E2 -15282.427} C_VEL
LIN {X 0,Y 326.538,Z 560.371,A -85,B 0,C 180,E1 -15283.752,E2 -15283.752} C_VEL
LIN {X 0,Y 324.816,Z 568.949,A -85,B 0,C 180,E1 -15285.272,E2 -15285.272} C_VEL
LIN {X 0,Y 323.301,Z 575.99,A -85,B 0,C 180,E1 -15286.806,E2 -15286.806} C_VEL
LIN {X 0,Y 321.768,Z 582.718,A -85,B 0,C 180,E1 -15288.663,E2 -15288.663} C_VEL
LIN {X 0,Y 320.911,Z 586.281,A -85,B 0,C 180,E1 -15289.91,E2 -15289.91} C_VEL
LIN {X 0,Y 320.242,Z 589.145,A -85,B 0,C 180,E1 -15291.163,E2 -15291.163} C_VEL
LIN {X 0,Y 319.425,Z 591.46,A -85,B 0,C 180,E1 -15292.414,E2 -15292.414} C_VEL
LIN {X 0,Y 319.058,Z 593.227,A -85,B 0,C 180,E1 -15293.677,E2 -15293.677} C_VEL
LIN {X 0,Y 318.889,Z 594.5,A -85,B 0,C 180,E1 -15294.943,E2 -15294.943} C_VEL
LIN {X 0,Y 318.532,Z 595.303,A -85,B 0,C 180,E1 -15296.205,E2 -15296.205} C_VEL
LIN {X 0,Y 318.245,Z 595.515,A -85,B 0,C 180,E1 -15297.469,E2 -15297.469} C_VEL
LIN {X 0,Y 318.029,Z 595.215,A -85,B 0,C 180,E1 -15298.734,E2 -15298.734} C_VEL
LIN {X 0,Y 317.942,Z 594.436,A -85,B 0,C 180,E1 -15300,E2 -15300} C_VEL
LIN {X 0,Y 317.904,Z 593.175,A -85,B 0,C 180,E1 -15301.267,E2 -15301.267} C_VEL
LIN {X 0,Y 318,Z 590.172,A -85,B 0,C 180,E1 -15303.167,E2 -15303.167} C_VEL
LIN {X 0,Y 318.212,Z 585.886,A -85,B 0,C 180,E1 -15305.068,E2 -15305.068} C_VEL
LIN {X 0,Y 318.475,Z 580.16,A -85,B 0,C 180,E1 -15306.971,E2 -15306.971} C_VEL
LIN {X 0,Y 318.854,Z 573.93,A -85,B 0,C 180,E1 -15308.556,E2 -15308.556} C_VEL
LIN {X 0,Y 319.247,Z 567.904,A -85,B 0,C 180,E1 -15309.823,E2 -15309.823} C_VEL
LIN {X 0,Y 319.858,Z 559.677,A -85,B 0,C 180,E1 -15311.245,E2 -15311.245} C_VEL
LIN {X 0,Y 320.462,Z 550.737,A -85,B 0,C 180,E1 -15312.508,E2 -15312.508} C_VEL
LIN {X 0,Y 321.075,Z 540.966,A -85,B 0,C 180,E1 -15313.61,E2 -15313.61} C_VEL
LIN {X 0,Y 321.318,Z 537.581,A -85,B 0,C 180,E1 -15313.922,E2 -15313.922} C_VEL
LIN {X 0,Y 319.825,Z 527.478,A -85,B 0,C 180,E1 -15314.785,E2 -15314.785} C_VEL
LIN {X 0,Y 318.19,Z 515.494,A -85,B 0,C 180,E1 -15315.575,E2 -15315.575} C_VEL
LIN {X 0,Y 318.222,Z 511.164,A -85,B 0,C 180,E1 -15319.346,E2 -15319.346} C_VEL
LIN {X 0,Y 318.358,Z 508.129,A -85,B 0,C 180,E1 -15322.042,E2 -15322.042} C_VEL
LIN {X 0,Y 318.53,Z 505.851,A -85,B 0,C 180,E1 -15324.264,E2 -15324.264} C_VEL
LIN {X 0,Y 319.748,Z 510.209,A -85,B 0,C 180,E1 -15326.781,E2 -15326.781} C_VEL
LIN {X 0,Y 319.68,Z 515.39,A -85,B 0,C 180,E1 -15329.647,E2 -15329.647} C_VEL
LIN {X 0,Y 319.351,Z 522.231,A -85,B 0,C 180,E1 -15333.379,E2 -15333.379} C_VEL
LIN {X 0,Y 319.053,Z 528.86,A -85,B 0,C 180,E1 -15337.015,E2 -15337.015} C_VEL
LIN {X 0,Y 318.999,Z 529.75,A -85,B 0,C 180,E1 -15337.505,E2 -15337.505} C_VEL
LIN {X 0,Y 321.556,Z 540.655,A -85,B 0,C 180,E1 -15338.229,E2 -15338.229} C_VEL
LIN {X 0,Y 323.354,Z 550.951,A -85,B 0,C 180,E1 -15339.073,E2 -15339.073} C_VEL
LIN {X 0,Y 324.053,Z 559.959,A -85,B 0,C 180,E1 -15339.964,E2 -15339.964} C_VEL
LIN {X 0,Y 323.1,Z 569.107,A -85,B 0,C 180,E1 -15341.011,E2 -15341.011} C_VEL
LIN {X 0,Y 322.143,Z 576.9,A -85,B 0,C 180,E1 -15342.118,E2 -15342.118} C_VEL
LIN {X 0,Y 321.222,Z 583.869,A -85,B 0,C 180,E1 -15343.327,E2 -15343.327} C_VEL
LIN {X 0,Y 320.449,Z 589.773,A -85,B 0,C 180,E1 -15344.573,E2 -15344.573} C_VEL
LIN {X 0,Y 319.679,Z 595.327,A -85,B 0,C 180,E1 -15346,E2 -15346} C_VEL
LIN {X 0,Y 318.982,Z 600.822,A -85,B 0,C 180,E1 -15347.779,E2 -15347.779} C_VEL
LIN {X 0,Y 318.455,Z 604.55,A -85,B 0,C 180,E1 -15349.379,E2 -15349.379} C_VEL
LIN {X 0,Y 318.178,Z 606.769,A -85,B 0,C 180,E1 -15350.632,E2 -15350.632} C_VEL
LIN {X 0,Y 317.761,Z 609.322,A -85,B 0,C 180,E1 -15352.771,E2 -15352.771} C_VEL
LIN {X 0,Y 317.575,Z 610.421,A -85,B 0,C 180,E1 -15354.967,E2 -15354.967} C_VEL
LIN {X 0,Y 317.564,Z 610.047,A -85,B 0,C 180,E1 -15357.244,E2 -15357.244} C_VEL
LIN {X 0,Y 317.802,Z 607.804,A -85,B 0,C 180,E1 -15359.594,E2 -15359.594} C_VEL
LIN {X 0,Y 318.024,Z 605.782,A -85,B 0,C 180,E1 -15360.91,E2 -15360.91} C_VEL
LIN {X 0,Y 318.268,Z 602.804,A -85,B 0,C 180,E1 -15362.372,E2 -15362.372} C_VEL
LIN {X 0,Y 318.622,Z 599.003,A -85,B 0,C 180,E1 -15363.822,E2 -15363.822} C_VEL
LIN {X 0,Y 319.132,Z 594.268,A -85,B 0,C 180,E1 -15365.264,E2 -15365.264} C_VEL
LIN {X 0,Y 319.743,Z 588.481,A -85,B 0,C 180,E1 -15366.693,E2 -15366.693} C_VEL
LIN {X 0,Y 320.428,Z 581.447,A -85,B 0,C 180,E1 -15368.107,E2 -15368.107} C_VEL
LIN {X 0,Y 321.324,Z 572.594,A -85,B 0,C 180,E1 -15369.515,E2 -15369.515} C_VEL
LIN {X 0,Y 322.101,Z 563.726,A -85,B 0,C 180,E1 -15370.619,E2 -15370.619} C_VEL
LIN {X 0,Y 322.59,Z 557.613,A -85,B 0,C 180,E1 -15371.255,E2 -15371.255} C_VEL
LIN {X 0,Y 321.67,Z 549.268,A -85,B 0,C 180,E1 -15372.024,E2 -15372.024} C_VEL
LIN {X 0,Y 320.149,Z 539.218,A -85,B 0,C 180,E1 -15372.761,E2 -15372.761} C_VEL
LIN {X 0,Y 318.43,Z 529.598,A -85,B 0,C 180,E1 -15373.326,E2 -15373.326} C_VEL
LIN {X 0,Y 318.714,Z 522.831,A -85,B 0,C 180,E1 -15377.26,E2 -15377.26} C_VEL
LIN {X 0,Y 319.006,Z 516.122,A -85,B 0,C 180,E1 -15381.128,E2 -15381.128} C_VEL
LIN {X 0,Y 319.289,Z 509.477,A -85,B 0,C 180,E1 -15384.948,E2 -15384.948} C_VEL
LIN {X 0,Y 319.446,Z 505.507,A -85,B 0,C 180,E1 -15387.399,E2 -15387.399} C_VEL
LIN {X 0,Y 320.049,Z 505.43,A -85,B 0,C 180,E1 -15389.999,E2 -15389.999} C_VEL
LIN {X 0,Y 319.993,Z 505.439,A -85,B 0,C 180,E1 -15392.517,E2 -15392.517} C_VEL
LIN {X 0,Y 319.954,Z 505.445,A -85,B 0,C 180,E1 -15396.305,E2 -15396.305} C_VEL
LIN {X 0,Y 319.843,Z 505.454,A -85,B 0,C 180,E1 -15398.847,E2 -15398.847} C_VEL
LIN {X 0,Y 319.683,Z 505.475,A -85,B 0,C 180,E1 -15402.699,E2 -15402.699} C_VEL
LIN {X 0,Y 319.7,Z 505.471,A -85,B 0,C 180,E1 -15405.295,E2 -15405.295} C_VEL
LIN {X 0,Y 319.675,Z 505.474,A -85,B 0,C 180,E1 -15409.254,E2 -15409.254} C_VEL
LIN {X 0,Y 319.57,Z 505.487,A -85,B 0,C 180,E1 -15413.319,E2 -15413.319} C_VEL
LIN {X 0,Y 319.635,Z 505.484,A -85,B 0,C 180,E1 -15416.087,E2 -15416.087} C_VEL
LIN {X 0,Y 319.597,Z 505.484,A -85,B 0,C 180,E1 -15418.932,E2 -15418.932} C_VEL
LIN {X 0,Y 319.532,Z 505.495,A -85,B 0,C 180,E1 -15421.861,E2 -15421.861} C_VEL
LIN {X 0,Y 319.579,Z 505.487,A -85,B 0,C 180,E1 -15425.542,E2 -15425.542} C_VEL
LIN {X 0,Y 319.572,Z 505.492,A -85,B 0,C 180,E1 -15428.007,E2 -15428.007} C_VEL
LIN {X 0,Y 319.562,Z 505.49,A -85,B 0,C 180,E1 -15431.604,E2 -15431.604} C_VEL
LIN {X 0,Y 319.579,Z 505.486,A -85,B 0,C 180,E1 -15435.273,E2 -15435.273} C_VEL
LIN {X 0,Y 319.577,Z 505.487,A -85,B 0,C 180,E1 -15438.719,E2 -15438.719} C_VEL
LIN {X 0,Y 319.596,Z 505.487,A -85,B 0,C 180,E1 -15442.339,E2 -15442.339} C_VEL
LIN {X 0,Y 319.557,Z 505.489,A -85,B 0,C 180,E1 -15445.123,E2 -15445.123} C_VEL
LIN {X 0,Y 319.567,Z 505.488,A -85,B 0,C 180,E1 -15449.058,E2 -15449.058} C_VEL
LIN {X 0,Y 319.605,Z 505.484,A -85,B 0,C 180,E1 -15452.498,E2 -15452.498} C_VEL
LIN {X 0,Y 319.605,Z 505.483,A -85,B 0,C 180,E1 -15454.866,E2 -15454.866} C_VEL
LIN {X 0,Y 318.915,Z 505.575,A -85,B 0,C 180,E1 -15455.918,E2 -15455.918} C_VEL
LIN {X 0,Y 316.034,Z 505.933,A -85,B 0,C 180,E1 -15457.628,E2 -15457.628} C_VEL
LIN {X 0,Y 313.636,Z 506.232,A -85,B 0,C 180,E1 -15459.015,E2 -15459.015} C_VEL
LIN {X 0,Y 312.654,Z 506.352,A -85,B 0,C 180,E1 -15460.089,E2 -15460.089} C_VEL
LIN {X 0,Y 312.599,Z 506.357,A -85,B 0,C 180,E1 -15460.453,E2 -15460.453} C_VEL
LIN {X 0,Y 312.636,Z 506.353,A -85,B 0,C 180,E1 -15464.35,E2 -15464.35} C_VEL
LIN {X 0,Y 312.634,Z 506.351,A -85,B 0,C 180,E1 -15467.009,E2 -15467.009} C_VEL
LIN {X 0,Y 312.831,Z 506.328,A -85,B 0,C 180,E1 -15471.296,E2 -15471.296} C_VEL
LIN {X 0,Y 312.908,Z 506.32,A -85,B 0,C 180,E1 -15473.552,E2 -15473.552} C_VEL
LIN {X 0,Y 312.936,Z 506.316,A -85,B 0,C 180,E1 -15477.426,E2 -15477.426} C_VEL
LIN {X 0,Y 313.1,Z 506.296,A -85,B 0,C 180,E1 -15480,E2 -15480} C_VEL
LIN {X 0,Y 312.936,Z 506.314,A -85,B 0,C 180,E1 -15482.574,E2 -15482.574} C_VEL
LIN {X 0,Y 312.908,Z 506.318,A -85,B 0,C 180,E1 -15486.448,E2 -15486.448} C_VEL
LIN {X 0,Y 312.785,Z 506.333,A -85,B 0,C 180,E1 -15489.049,E2 -15489.049} C_VEL
LIN {X 0,Y 312.631,Z 506.352,A -85,B 0,C 180,E1 -15492.991,E2 -15492.991} C_VEL
LIN {X 0,Y 312.635,Z 506.357,A -85,B 0,C 180,E1 -15495.65,E2 -15495.65} C_VEL
LIN {X 0,Y 312.627,Z 506.354,A -85,B 0,C 180,E1 -15499.236,E2 -15499.236} C_VEL
LIN {X 0,Y 312.543,Z 506.363,A -85,B 0,C 180,E1 -15502.789,E2 -15502.789} C_VEL
LIN {X 0,Y 312.6,Z 506.358,A -85,B 0,C 180,E1 -15505.936,E2 -15505.936} C_VEL
LIN {X 0,Y 312.543,Z 506.368,A -85,B 0,C 180,E1 -15509.65,E2 -15509.65} C_VEL
LIN {X 0,Y 312.517,Z 506.37,A -85,B 0,C 180,E1 -15513.689,E2 -15513.689} C_VEL
LIN {X 0,Y 312.535,Z 506.368,A -85,B 0,C 180,E1 -15517.384,E2 -15517.384} C_VEL
LIN {X 0,Y 312.487,Z 506.37,A -85,B 0,C 180,E1 -15520.709,E2 -15520.709} C_VEL
LIN {X 0,Y 312.473,Z 506.372,A -85,B 0,C 180,E1 -15524.206,E2 -15524.206} C_VEL
LIN {X 0,Y 312.53,Z 506.366,A -85,B 0,C 180,E1 -15527.909,E2 -15527.909} C_VEL
LIN {X 0,Y 312.686,Z 506.488,A -85,B 0,C 180,E1 -15532.262,E2 -15532.262} C_VEL
LIN {X 0,Y 313.732,Z 512.496,A -85,B 0,C 180,E1 -15535.98,E2 -15535.98} C_VEL
LIN {X 0,Y 314.148,Z 515.067,A -85,B 0,C 180,E1 -15537.527,E2 -15537.527} C_VEL
LIN {X 0,Y 313.612,Z 520.169,A -85,B 0,C 180,E1 -15540.462,E2 -15540.462} C_VEL
LIN {X 0,Y 312.767,Z 526.438,A -85,B 0,C 180,E1 -15544.003,E2 -15544.003} C_VEL
LIN {X 0,Y 312.079,Z 532.695,A -85,B 0,C 180,E1 -15547.491,E2 -15547.491} C_VEL
LIN {X 0,Y 311.448,Z 540.053,A -85,B 0,C 180,E1 -15551.584,E2 -15551.584} C_VEL
LIN {X 0,Y 311.362,Z 541.64,A -85,B 0,C 180,E1 -15552.471,E2 -15552.471} C_VEL
LIN {X 0,Y 312.886,Z 554.405,A -85,B 0,C 180,E1 -15553.069,E2 -15553.069} C_VEL
LIN {X 0,Y 313.756,Z 564.243,A -85,B 0,C 180,E1 -15553.716,E2 -15553.716} C_VEL
LIN {X 0,Y 314.369,Z 574.555,A -85,B 0,C 180,E1 -15554.605,E2 -15554.605} C_VEL
LIN {X 0,Y 314.402,Z 582.204,A -85,B 0,C 180,E1 -15555.436,E2 -15555.436} C_VEL
LIN {X 0,Y 313.463,Z 591.802,A -85,B 0,C 180,E1 -15556.715,E2 -15556.715} C_VEL
LIN {X 0,Y 312.734,Z 599.429,A -85,B 0,C 180,E1 -15558.003,E2 -15558.003} C_VEL
LIN {X 0,Y 312.109,Z 605.686,A -85,B 0,C 180,E1 -15559.295,E2 -15559.295} C_VEL
LIN {X 0,Y 311.635,Z 610.869,A -85,B 0,C 180,E1 -15560.59,E2 -15560.59} C_VEL
LIN {X 0,Y 311.18,Z 616.126,A -85,B 0,C 180,E1 -15562.213,E2 -15562.213} C_VEL
LIN {X 0,Y 310.835,Z 621.015,A -85,B 0,C 180,E1 -15564.178,E2 -15564.178} C_VEL
LIN {X 0,Y 310.8,Z 624.3,A -85,B 0,C 180,E1 -15566.111,E2 -15566.111} C_VEL
LIN {X 0,Y 310.731,Z 625.866,A -85,B 0,C 180,E1 -15567.408,E2 -15567.408} C_VEL
LIN {X 0,Y 310.701,Z 626.829,A -85,B 0,C 180,E1 -15568.705,E2 -15568.705} C_VEL
LIN {X 0,Y 310.751,Z 627.256,A -85,B 0,C 180,E1 -15570.001,E2 -15570.001} C_VEL
LIN {X 0,Y 310.698,Z 627.195,A -85,B 0,C 180,E1 -15571.297,E2 -15571.297} C_VEL
LIN {X 0,Y 310.725,Z 626.653,A -85,B 0,C 180,E1 -15572.593,E2 -15572.593} C_VEL
LIN {X 0,Y 310.779,Z 625.61,A -85,B 0,C 180,E1 -15573.891,E2 -15573.891} C_VEL
LIN {X 0,Y 310.886,Z 622.782,A -85,B 0,C 180,E1 -15575.914,E2 -15575.914} C_VEL
LIN {X 0,Y 311.674,Z 617.164,A -85,B 0,C 180,E1 -15579.082,E2 -15579.082} C_VEL
LIN {X 0,Y 312.639,Z 612.306,A -85,B 0,C 180,E1 -15581.016,E2 -15581.016} C_VEL
LIN {X 0,Y 313.701,Z 607.134,A -85,B 0,C 180,E1 -15582.618,E2 -15582.618} C_VEL
LIN {X 0,Y 315.089,Z 600.809,A -85,B 0,C 180,E1 -15584.203,E2 -15584.203} C_VEL
LIN {X 0,Y 316.596,Z 593.199,A -85,B 0,C 180,E1 -15585.78,E2 -15585.78} C_VEL
LIN {X 0,Y 318.099,Z 585.841,A -85,B 0,C 180,E1 -15587.023,E2 -15587.023} C_VEL
LIN {X 0,Y 318.954,Z 577.038,A -85,B 0,C 180,E1 -15588.335,E2 -15588.335} C_VEL
LIN {X 0,Y 318.761,Z 568.564,A -85,B 0,C 180,E1 -15589.505,E2 -15589.505} C_VEL
LIN {X 0,Y 317.49,Z 559.047,A -85,B 0,C 180,E1 -15590.744,E2 -15590.744} C_VEL
LIN {X 0,Y 315.051,Z 548.277,A -85,B 0,C 180,E1 -15592.114,E2 -15592.114} C_VEL
LIN {X 0,Y 312.689,Z 540.698,A -85,B 0,C 180,E1 -15593.078,E2 -15593.078} C_VEL
LIN {X 0,Y 312.644,Z 539.938,A -85,B 0,C 180,E1 -15593.239,E2 -15593.239} C_VEL
LIN {X 0,Y 313.474,Z 535.041,A -85,B 0,C 180,E1 -15596.641,E2 -15596.641} C_VEL
LIN {X 0,Y 314.271,Z 531.279,A -85,B 0,C 180,E1 -15599.472,E2 -15599.472} C_VEL
LIN {X 0,Y 315.046,Z 527.781,A -85,B 0,C 180,E1 -15602.371,E2 -15602.371} C_VEL
LIN {X 0,Y 315.435,Z 525.529,A -85,B 0,C 180,E1 -15604.475,E2 -15604.475} C_VEL
LIN {X 0,Y 315.425,Z 523.254,A -85,B 0,C 180,E1 -15606.985,E2 -15606.985} C_VEL
LIN {X 0,Y 315.076,Z 520.837,A -85,B 0,C 180,E1 -15610.307,E2 -15610.307} C_VEL
LIN {X 0,Y 314.791,Z 518.956,A -85,B 0,C 180,E1 -15613.798,E2 -15613.798} C_VEL
LIN {X 0,Y 314.565,Z 517.696,A -85,B 0,C 180,E1 -15617.502,E2 -15617.502} C_VEL
LIN {X 0,Y 314.398,Z 517.144,A -85,B 0,C 180,E1 -15621.48,E2 -15621.48} C_VEL
LIN {X 0,Y 314.301,Z 517.231,A -85,B 0,C 180,E1 -15624.453,E2 -15624.453} C_VEL
LIN {X 0,Y 314.11,Z 517.766,A -85,B 0,C 180,E1 -15627.522,E2 -15627.522} C_VEL
LIN {X 0,Y 313.648,Z 518.839,A -85,B 0,C 180,E1 -15630.914,E2 -15630.914} C_VEL
LIN {X 0,Y 313.066,Z 520.561,A -85,B 0,C 180,E1 -15634.753,E2 -15634.753} C_VEL
LIN {X 0,Y 312.811,Z 521.935,A -85,B 0,C 180,E1 -15637.042,E2 -15637.042} C_VEL
LIN {X 0,Y 313.451,Z 523.972,A -85,B 0,C 180,E1 -15637.318,E2 -15637.318} C_VEL
LIN {X 0,Y 314.556,Z 525.847,A -85,B 0,C 180,E1 -15637.677,E2 -15637.677} C_VEL
LIN {X 0,Y 318.187,Z 534.844,A -85,B 0,C 180,E1 -15639.135,E2 -15639.135} C_VEL
LIN {X 0,Y 320.656,Z 543.257,A -85,B 0,C 180,E1 -15640.47,E2 -15640.47} C_VEL
LIN {X 0,Y 322.008,Z 550.624,A -85,B 0,C 180,E1 -15641.66,E2 -15641.66} C_VEL
LIN {X 0,Y 321.826,Z 553.213,A -85,B 0,C 180,E1 -15642.015,E2 -15642.015} C_VEL
LIN {X 0,Y 319.964,Z 562.535,A -85,B 0,C 180,E1 -15643.409,E2 -15643.409} C_VEL
LIN {X 0,Y 318.515,Z 569.317,A -85,B 0,C 180,E1 -15644.646,E2 -15644.646} C_VEL
LIN {X 0,Y 317.146,Z 575.034,A -85,B 0,C 180,E1 -15645.891,E2 -15645.891} C_VEL
LIN {X 0,Y 315.696,Z 580.926,A -85,B 0,C 180,E1 -15647.464,E2 -15647.464} C_VEL
LIN {X 0,Y 314.432,Z 585.707,A -85,B 0,C 180,E1 -15649.048,E2 -15649.048} C_VEL
LIN {X 0,Y 313.299,Z 590.161,A -85,B 0,C 180,E1 -15650.966,E2 -15650.966} C_VEL
LIN {X 0,Y 312.445,Z 592.352,A -85,B 0,C 180,E1 -15652.244,E2 -15652.244} C_VEL
LIN {X 0,Y 312.035,Z 593.962,A -85,B 0,C 180,E1 -15653.534,E2 -15653.534} C_VEL
LIN {X 0,Y 311.83,Z 595.084,A -85,B 0,C 180,E1 -15654.828,E2 -15654.828} C_VEL
LIN {X 0,Y 311.463,Z 595.769,A -85,B 0,C 180,E1 -15656.119,E2 -15656.119} C_VEL
LIN {X 0,Y 311.166,Z 595.944,A -85,B 0,C 180,E1 -15657.411,E2 -15657.411} C_VEL
LIN {X 0,Y 310.938,Z 595.525,A -85,B 0,C 180,E1 -15658.705,E2 -15658.705} C_VEL
LIN {X 0,Y 310.846,Z 594.617,A -85,B 0,C 180,E1 -15660,E2 -15660} C_VEL
LIN {X 0,Y 310.813,Z 593.22,A -85,B 0,C 180,E1 -15661.296,E2 -15661.296} C_VEL
LIN {X 0,Y 310.928,Z 590.083,A -85,B 0,C 180,E1 -15663.24,E2 -15663.24} C_VEL
LIN {X 0,Y 311.073,Z 587.27,A -85,B 0,C 180,E1 -15664.535,E2 -15664.535} C_VEL
LIN {X 0,Y 311.161,Z 583.352,A -85,B 0,C 180,E1 -15665.99,E2 -15665.99} C_VEL
LIN {X 0,Y 311.547,Z 578.497,A -85,B 0,C 180,E1 -15667.453,E2 -15667.453} C_VEL
LIN {X 0,Y 311.811,Z 573.282,A -85,B 0,C 180,E1 -15668.751,E2 -15668.751} C_VEL
LIN {X 0,Y 312.241,Z 567.068,A -85,B 0,C 180,E1 -15670.046,E2 -15670.046} C_VEL
LIN {X 0,Y 312.794,Z 559.627,A -85,B 0,C 180,E1 -15671.338,E2 -15671.338} C_VEL
LIN {X 0,Y 313.404,Z 550.616,A -85,B 0,C 180,E1 -15672.629,E2 -15672.629} C_VEL
LIN {X 0,Y 314.037,Z 540.651,A -85,B 0,C 180,E1 -15673.756,E2 -15673.756} C_VEL
LIN {X 0,Y 314.15,Z 537.237,A -85,B 0,C 180,E1 -15674.081,E2 -15674.081} C_VEL
LIN {X 0,Y 312.481,Z 526.404,A -85,B 0,C 180,E1 -15675.015,E2 -15675.015} C_VEL
LIN {X 0,Y 311.084,Z 515.802,A -85,B 0,C 180,E1 -15675.73,E2 -15675.73} C_VEL
LIN {X 0,Y 311.171,Z 512.71,A -85,B 0,C 180,E1 -15678.449,E2 -15678.449} C_VEL
LIN {X 0,Y 311.28,Z 508.134,A -85,B 0,C 180,E1 -15682.571,E2 -15682.571} C_VEL
LIN {X 0,Y 311.392,Z 506.765,A -85,B 0,C 180,E1 -15683.926,E2 -15683.926} C_VEL
LIN {X 0,Y 312.744,Z 511.433,A -85,B 0,C 180,E1 -15686.708,E2 -15686.708} C_VEL
LIN {X 0,Y 312.798,Z 515.185,A -85,B 0,C 180,E1 -15688.804,E2 -15688.804} C_VEL
LIN {X 0,Y 312.399,Z 522.139,A -85,B 0,C 180,E1 -15692.679,E2 -15692.679} C_VEL
LIN {X 0,Y 312.061,Z 529.639,A -85,B 0,C 180,E1 -15696.843,E2 -15696.843} C_VEL
LIN {X 0,Y 312.043,Z 529.912,A -85,B 0,C 180,E1 -15696.997,E2 -15696.997} C_VEL
LIN {X 0,Y 314.592,Z 540.586,A -85,B 0,C 180,E1 -15697.731,E2 -15697.731} C_VEL
LIN {X 0,Y 316.479,Z 551.214,A -85,B 0,C 180,E1 -15698.633,E2 -15698.633} C_VEL
LIN {X 0,Y 317.264,Z 560.893,A -85,B 0,C 180,E1 -15699.634,E2 -15699.634} C_VEL
LIN {X 0,Y 316.283,Z 569.722,A -85,B 0,C 180,E1 -15700.678,E2 -15700.678} C_VEL
LIN {X 0,Y 315.299,Z 577.391,A -85,B 0,C 180,E1 -15701.798,E2 -15701.798} C_VEL
LIN {X 0,Y 314.284,Z 584.746,A -85,B 0,C 180,E1 -15703.117,E2 -15703.117} C_VEL
LIN {X 0,Y 313.354,Z 591.411,A -85,B 0,C 180,E1 -15704.593,E2 -15704.593} C_VEL
LIN {X 0,Y 312.425,Z 597.72,A -85,B 0,C 180,E1 -15706.376,E2 -15706.376} C_VEL
LIN {X 0,Y 311.802,Z 602.269,A -85,B 0,C 180,E1 -15708.058,E2 -15708.058} C_VEL
LIN {X 0,Y 311.437,Z 604.663,A -85,B 0,C 180,E1 -15709.123,E2 -15709.123} C_VEL
LIN {X 0,Y 311.053,Z 607.434,A -85,B 0,C 180,E1 -15710.754,E2 -15710.754} C_VEL
LIN {X 0,Y 310.739,Z 609.317,A -85,B 0,C 180,E1 -15712.362,E2 -15712.362} C_VEL
LIN {X 0,Y 310.49,Z 610.545,A -85,B 0,C 180,E1 -15714.574,E2 -15714.574} C_VEL
LIN {X 0,Y 310.439,Z 610.722,A -85,B 0,C 180,E1 -15715.529,E2 -15715.529} C_VEL
LIN {X 0,Y 310.454,Z 610.308,A -85,B 0,C 180,E1 -15717.09,E2 -15717.09} C_VEL
LIN {X 0,Y 310.65,Z 608.415,A -85,B 0,C 180,E1 -15719.282,E2 -15719.282} C_VEL
LIN {X 0,Y 310.946,Z 606.041,A -85,B 0,C 180,E1 -15720.925,E2 -15720.925} C_VEL
LIN {X 0,Y 311.217,Z 602.961,A -85,B 0,C 180,E1 -15722.473,E2 -15722.473} C_VEL
LIN {X 0,Y 311.532,Z 599.498,A -85,B 0,C 180,E1 -15723.837,E2 -15723.837} C_VEL
LIN {X 0,Y 312.091,Z 594.59,A -85,B 0,C 180,E1 -15725.379,E2 -15725.379} C_VEL
LIN {X 0,Y 312.61,Z 589.599,A -85,B 0,C 180,E1 -15726.662,E2 -15726.662} C_VEL
LIN {X 0,Y 313.212,Z 583.701,A -85,B 0,C 180,E1 -15727.923,E2 -15727.923} C_VEL
LIN {X 0,Y 314.005,Z 576.159,A -85,B 0,C 180,E1 -15729.244,E2 -15729.244} C_VEL
LIN {X 0,Y 314.959,Z 566.364,A -85,B 0,C 180,E1 -15730.614,E2 -15730.614} C_VEL
LIN {X 0,Y 315.633,Z 558.223,A -85,B 0,C 180,E1 -15731.5,E2 -15731.5} C_VEL
LIN {X 0,Y 314.725,Z 549.966,A -85,B 0,C 180,E1 -15732.286,E2 -15732.286} C_VEL
LIN {X 0,Y 313.222,Z 540.024,A -85,B 0,C 180,E1 -15733.04,E2 -15733.04} C_VEL
LIN {X 0,Y 311.512,Z 530.811,A -85,B 0,C 180,E1 -15733.577,E2 -15733.577} C_VEL
LIN {X 0,Y 311.386,Z 529.746,A -85,B 0,C 180,E1 -15733.654,E2 -15733.654} C_VEL
LIN {X 0,Y 311.674,Z 522.999,A -85,B 0,C 180,E1 -15737.63,E2 -15737.63} C_VEL
LIN {X 0,Y 311.969,Z 516.256,A -85,B 0,C 180,E1 -15741.579,E2 -15741.579} C_VEL
LIN {X 0,Y 312.278,Z 509.601,A -85,B 0,C 180,E1 -15745.482,E2 -15745.482} C_VEL
LIN {X 0,Y 312.376,Z 506.388,A -85,B 0,C 180,E1 -15747.42,E2 -15747.42} C_VEL
LIN {X 0,Y 313.006,Z 506.308,A -85,B 0,C 180,E1 -15749.999,E2 -15749.999} C_VEL
LIN {X 0,Y 312.939,Z 506.317,A -85,B 0,C 180,E1 -15752.574,E2 -15752.574} C_VEL
LIN {X 0,Y 312.912,Z 506.321,A -85,B 0,C 180,E1 -15756.447,E2 -15756.447} C_VEL
LIN {X 0,Y 312.789,Z 506.333,A -85,B 0,C 180,E1 -15759.048,E2 -15759.048} C_VEL
LIN {X 0,Y 312.635,Z 506.352,A -85,B 0,C 180,E1 -15762.99,E2 -15762.99} C_VEL
LIN {X 0,Y 312.639,Z 506.352,A -85,B 0,C 180,E1 -15765.649,E2 -15765.649} C_VEL
LIN {X 0,Y 312.631,Z 506.352,A -85,B 0,C 180,E1 -15769.236,E2 -15769.236} C_VEL
LIN {X 0,Y 312.546,Z 506.363,A -85,B 0,C 180,E1 -15772.789,E2 -15772.789} C_VEL
LIN {X 0,Y 312.603,Z 506.358,A -85,B 0,C 180,E1 -15775.935,E2 -15775.935} C_VEL
LIN {X 0,Y 312.548,Z 506.363,A -85,B 0,C 180,E1 -15779.649,E2 -15779.649} C_VEL
LIN {X 0,Y 312.518,Z 506.367,A -85,B 0,C 180,E1 -15783.688,E2 -15783.688} C_VEL
LIN {X 0,Y 312.536,Z 506.364,A -85,B 0,C 180,E1 -15787.383,E2 -15787.383} C_VEL
LIN {X 0,Y 312.494,Z 506.369,A -85,B 0,C 180,E1 -15790.708,E2 -15790.708} C_VEL
LIN {X 0,Y 312.527,Z 506.369,A -85,B 0,C 180,E1 -15794.195,E2 -15794.195} C_VEL
LIN {X 0,Y 312.547,Z 506.366,A -85,B 0,C 180,E1 -15797.905,E2 -15797.905} C_VEL
LIN {X 0,Y 312.556,Z 506.365,A -85,B 0,C 180,E1 -15801.904,E2 -15801.904} C_VEL
LIN {X 0,Y 312.504,Z 506.371,A -85,B 0,C 180,E1 -15805.789,E2 -15805.789} C_VEL
LIN {X 0,Y 312.521,Z 506.366,A -85,B 0,C 180,E1 -15808.854,E2 -15808.854} C_VEL
LIN {X 0,Y 312.571,Z 506.363,A -85,B 0,C 180,E1 -15811.824,E2 -15811.824} C_VEL
LIN {X 0,Y 312.57,Z 506.359,A -85,B 0,C 180,E1 -15814.847,E2 -15814.847} C_VEL
LIN {X 0,Y 312.585,Z 506.36,A -85,B 0,C 180,E1 -15817.529,E2 -15817.529} C_VEL
LIN {X 0,Y 312.599,Z 506.357,A -85,B 0,C 180,E1 -15820.453,E2 -15820.453} C_VEL
LIN {X 0,Y 312.001,Z 506.434,A -85,B 0,C 180,E1 -15821.529,E2 -15821.529} C_VEL
LIN {X 0,Y 309.183,Z 506.782,A -85,B 0,C 180,E1 -15823.28,E2 -15823.28} C_VEL
LIN {X 0,Y 306.745,Z 507.085,A -85,B 0,C 180,E1 -15824.701,E2 -15824.701} C_VEL
LIN {X 0,Y 305.683,Z 507.222,A -85,B 0,C 180,E1 -15825.801,E2 -15825.801} C_VEL
LIN {X 0,Y 305.591,Z 507.227,A -85,B 0,C 180,E1 -15826.174,E2 -15826.174} C_VEL
LIN {X 0,Y 305.733,Z 507.211,A -85,B 0,C 180,E1 -15830.74,E2 -15830.74} C_VEL
LIN {X 0,Y 305.85,Z 507.198,A -85,B 0,C 180,E1 -15833.402,E2 -15833.402} C_VEL
LIN {X 0,Y 305.957,Z 507.182,A -85,B 0,C 180,E1 -15838.684,E2 -15838.684} C_VEL
LIN {X 0,Y 305.955,Z 507.185,A -85,B 0,C 180,E1 -15841.316,E2 -15841.316} C_VEL
LIN {X 0,Y 305.85,Z 507.196,A -85,B 0,C 180,E1 -15846.597,E2 -15846.597} C_VEL
LIN {X 0,Y 305.733,Z 507.213,A -85,B 0,C 180,E1 -15849.26,E2 -15849.26} C_VEL
LIN {X 0,Y 305.586,Z 507.231,A -85,B 0,C 180,E1 -15853.296,E2 -15853.296} C_VEL
LIN {X 0,Y 305.591,Z 507.231,A -85,B 0,C 180,E1 -15856.02,E2 -15856.02} C_VEL
LIN {X 0,Y 305.573,Z 507.235,A -85,B 0,C 180,E1 -15859.445,E2 -15859.445} C_VEL
LIN {X 0,Y 305.488,Z 507.243,A -85,B 0,C 180,E1 -15863.042,E2 -15863.042} C_VEL
LIN {X 0,Y 305.545,Z 507.236,A -85,B 0,C 180,E1 -15866.227,E2 -15866.227} C_VEL
LIN {X 0,Y 305.493,Z 507.242,A -85,B 0,C 180,E1 -15869.05,E2 -15869.05} C_VEL
LIN {X 0,Y 305.445,Z 507.249,A -85,B 0,C 180,E1 -15871.952,E2 -15871.952} C_VEL
LIN {X 0,Y 305.46,Z 507.247,A -85,B 0,C 180,E1 -15875.113,E2 -15875.113} C_VEL
LIN {X 0,Y 305.464,Z 507.244,A -85,B 0,C 180,E1 -15878.533,E2 -15878.533} C_VEL
LIN {X 0,Y 305.475,Z 507.243,A -85,B 0,C 180,E1 -15882.591,E2 -15882.591} C_VEL
LIN {X 0,Y 305.478,Z 507.243,A -85,B 0,C 180,E1 -15886.355,E2 -15886.355} C_VEL
LIN {X 0,Y 305.468,Z 507.246,A -85,B 0,C 180,E1 -15889.895,E2 -15889.895} C_VEL
LIN {X 0,Y 305.661,Z 507.422,A -85,B 0,C 180,E1 -15892.253,E2 -15892.253} C_VEL
LIN {X 0,Y 306.582,Z 512.717,A -85,B 0,C 180,E1 -15895.614,E2 -15895.614} C_VEL
LIN {X 0,Y 307.061,Z 516.999,A -85,B 0,C 180,E1 -15898.237,E2 -15898.237} C_VEL
LIN {X 0,Y 306.154,Z 523.305,A -85,B 0,C 180,E1 -15901.928,E2 -15901.928} C_VEL
LIN {X 0,Y 305.236,Z 530.792,A -85,B 0,C 180,E1 -15906.239,E2 -15906.239} C_VEL
LIN {X 0,Y 304.549,Z 538.16,A -85,B 0,C 180,E1 -15910.452,E2 -15910.452} C_VEL
LIN {X 0,Y 304.284,Z 541.263,A -85,B 0,C 180,E1 -15912.137,E2 -15912.137} C_VEL
LIN {X 0,Y 305.747,Z 553.258,A -85,B 0,C 180,E1 -15912.679,E2 -15912.679} C_VEL
LIN {X 0,Y 306.635,Z 562.316,A -85,B 0,C 180,E1 -15913.267,E2 -15913.267} C_VEL
LIN {X 0,Y 307.173,Z 570.381,A -85,B 0,C 180,E1 -15913.934,E2 -15913.934} C_VEL
LIN {X 0,Y 307.521,Z 578.554,A -85,B 0,C 180,E1 -15914.769,E2 -15914.769} C_VEL
LIN {X 0,Y 307.142,Z 585.401,A -85,B 0,C 180,E1 -15915.592,E2 -15915.592} C_VEL
LIN {X 0,Y 306.325,Z 593.28,A -85,B 0,C 180,E1 -15916.737,E2 -15916.737} C_VEL
LIN {X 0,Y 305.57,Z 600.63,A -85,B 0,C 180,E1 -15918.054,E2 -15918.054} C_VEL
LIN {X 0,Y 304.809,Z 608.061,A -85,B 0,C 180,E1 -15919.707,E2 -15919.707} C_VEL
LIN {X 0,Y 304.295,Z 613.853,A -85,B 0,C 180,E1 -15921.367,E2 -15921.367} C_VEL
LIN {X 0,Y 303.969,Z 617.622,A -85,B 0,C 180,E1 -15922.695,E2 -15922.695} C_VEL
LIN {X 0,Y 303.704,Z 621.886,A -85,B 0,C 180,E1 -15924.69,E2 -15924.69} C_VEL
LIN {X 0,Y 303.712,Z 624.038,A -85,B 0,C 180,E1 -15926.02,E2 -15926.02} C_VEL
LIN {X 0,Y 303.656,Z 625.62,A -85,B 0,C 180,E1 -15927.348,E2 -15927.348} C_VEL
LIN {X 0,Y 303.616,Z 626.594,A -85,B 0,C 180,E1 -15928.674,E2 -15928.674} C_VEL
LIN {X 0,Y 303.661,Z 627.05,A -85,B 0,C 180,E1 -15930.001,E2 -15930.001} C_VEL
LIN {X 0,Y 303.613,Z 627.018,A -85,B 0,C 180,E1 -15931.327,E2 -15931.327} C_VEL
LIN {X 0,Y 303.649,Z 626.505,A -85,B 0,C 180,E1 -15932.654,E2 -15932.654} C_VEL
LIN {X 0,Y 303.694,Z 625.482,A -85,B 0,C 180,E1 -15933.982,E2 -15933.982} C_VEL
LIN {X 0,Y 303.785,Z 623.059,A -85,B 0,C 180,E1 -15935.85,E2 -15935.85} C_VEL
LIN {X 0,Y 304.657,Z 617.279,A -85,B 0,C 180,E1 -15939.293,E2 -15939.293} C_VEL
LIN {X 0,Y 305.676,Z 612.701,A -85,B 0,C 180,E1 -15941.27,E2 -15941.27} C_VEL
LIN {X 0,Y 307.088,Z 606.627,A -85,B 0,C 180,E1 -15943.231,E2 -15943.231} C_VEL
LIN {X 0,Y 308.616,Z 600.331,A -85,B 0,C 180,E1 -15944.845,E2 -15944.845} C_VEL
LIN {X 0,Y 309.842,Z 594.345,A -85,B 0,C 180,E1 -15946.133,E2 -15946.133} C_VEL
LIN {X 0,Y 311.452,Z 587.296,A -85,B 0,C 180,E1 -15947.398,E2 -15947.398} C_VEL
LIN {X 0,Y 312.464,Z 579.4,A -85,B 0,C 180,E1 -15948.665,E2 -15948.665} C_VEL
LIN {X 0,Y 312.466,Z 570.632,A -85,B 0,C 180,E1 -15949.97,E2 -15949.97} C_VEL
LIN {X 0,Y 311.402,Z 561.012,A -85,B 0,C 180,E1 -15951.342,E2 -15951.342} C_VEL
LIN {X 0,Y 309.224,Z 550.936,A -85,B 0,C 180,E1 -15952.73,E2 -15952.73} C_VEL
LIN {X 0,Y 307.141,Z 543.743,A -85,B 0,C 180,E1 -15953.755,E2 -15953.755} C_VEL
LIN {X 0,Y 305.973,Z 540.369,A -85,B 0,C 180,E1 -15954.224,E2 -15954.224} C_VEL
LIN {X 0,Y 305.873,Z 539.451,A -85,B 0,C 180,E1 -15954.332,E2 -15954.332} C_VEL
LIN {X 0,Y 306.614,Z 535.4,A -85,B 0,C 180,E1 -15957.286,E2 -15957.286} C_VEL
LIN {X 0,Y 307.444,Z 531.727,A -85,B 0,C 180,E1 -15960.193,E2 -15960.193} C_VEL
LIN {X 0,Y 308.231,Z 528.342,A -85,B 0,C 180,E1 -15963.178,E2 -15963.178} C_VEL
LIN {X 0,Y 308.491,Z 526.612,A -85,B 0,C 180,E1 -15964.901,E2 -15964.901} C_VEL
LIN {X 0,Y 308.369,Z 524.02,A -85,B 0,C 180,E1 -15967.978,E2 -15967.978} C_VEL
LIN {X 0,Y 308.046,Z 521.771,A -85,B 0,C 180,E1 -15971.425,E2 -15971.425} C_VEL
LIN {X 0,Y 307.769,Z 520.078,A -85,B 0,C 180,E1 -15975.065,E2 -15975.065} C_VEL
LIN {X 0,Y 307.578,Z 519.114,A -85,B 0,C 180,E1 -15978.499,E2 -15978.499} C_VEL
LIN {X 0,Y 307.449,Z 518.732,A -85,B 0,C 180,E1 -15981.889,E2 -15981.889} C_VEL
LIN {X 0,Y 307.337,Z 518.9,A -85,B 0,C 180,E1 -15985.41,E2 -15985.41} C_VEL
LIN {X 0,Y 307.124,Z 519.453,A -85,B 0,C 180,E1 -15988.243,E2 -15988.243} C_VEL
LIN {X 0,Y 306.637,Z 520.416,A -85,B 0,C 180,E1 -15991.229,E2 -15991.229} C_VEL
LIN {X 0,Y 306.177,Z 521.638,A -85,B 0,C 180,E1 -15994.143,E2 -15994.143} C_VEL
LIN {X 0,Y 305.93,Z 522.481,A -85,B 0,C 180,E1 -15995.847,E2 -15995.847} C_VEL
LIN {X 0,Y 307.01,Z 525.399,A -85,B 0,C 180,E1 -15996.303,E2 -15996.303} C_VEL
LIN {X 0,Y 308.297,Z 527.963,A -85,B 0,C 180,E1 -15996.8,E2 -15996.8} C_VEL
LIN {X 0,Y 311.616,Z 535.725,A -85,B 0,C 180,E1 -15998.218,E2 -15998.218} C_VEL
LIN {X 0,Y 314.195,Z 543.99,A -85,B 0,C 180,E1 -15999.652,E2 -15999.652} C_VEL
LIN {X 0,Y 315.759,Z 552.612,A -85,B 0,C 180,E1 -16001.13,E2 -16001.13} C_VEL
LIN {X 0,Y 315.412,Z 555.669,A -85,B 0,C 180,E1 -16001.586,E2 -16001.586} C_VEL
LIN {X 0,Y 313.804,Z 563.058,A -85,B 0,C 180,E1 -16002.738,E2 -16002.738} C_VEL
LIN {X 0,Y 311.87,Z 571.252,A -85,B 0,C 180,E1 -16004.311,E2 -16004.311} C_VEL
LIN {X 0,Y 309.843,Z 579.165,A -85,B 0,C 180,E1 -16006.222,E2 -16006.222} C_VEL
LIN {X 0,Y 308.644,Z 583.435,A -85,B 0,C 180,E1 -16007.507,E2 -16007.507} C_VEL
LIN {X 0,Y 307.133,Z 588.446,A -85,B 0,C 180,E1 -16009.452,E2 -16009.452} C_VEL
LIN {X 0,Y 305.874,Z 592.166,A -85,B 0,C 180,E1 -16011.411,E2 -16011.411} C_VEL
LIN {X 0,Y 305.465,Z 593.223,A -85,B 0,C 180,E1 -16012.065,E2 -16012.065} C_VEL
LIN {X 0,Y 305.016,Z 594.71,A -85,B 0,C 180,E1 -16013.385,E2 -16013.385} C_VEL
LIN {X 0,Y 304.774,Z 595.691,A -85,B 0,C 180,E1 -16014.708,E2 -16014.708} C_VEL
LIN {X 0,Y 304.394,Z 596.229,A -85,B 0,C 180,E1 -16016.028,E2 -16016.028} C_VEL
LIN {X 0,Y 304.083,Z 596.306,A -85,B 0,C 180,E1 -16017.351,E2 -16017.351} C_VEL
LIN {X 0,Y 303.847,Z 595.831,A -85,B 0,C 180,E1 -16018.675,E2 -16018.675} C_VEL
LIN {X 0,Y 303.752,Z 594.79,A -85,B 0,C 180,E1 -16020,E2 -16020} C_VEL
LIN {X 0,Y 303.739,Z 592.361,A -85,B 0,C 180,E1 -16021.989,E2 -16021.989} C_VEL
LIN {X 0,Y 303.931,Z 588.613,A -85,B 0,C 180,E1 -16023.978,E2 -16023.978} C_VEL
LIN {X 0,Y 304.055,Z 583.567,A -85,B 0,C 180,E1 -16025.918,E2 -16025.918} C_VEL
LIN {X 0,Y 304.499,Z 577.906,A -85,B 0,C 180,E1 -16027.626,E2 -16027.626} C_VEL
LIN {X 0,Y 304.862,Z 571.087,A -85,B 0,C 180,E1 -16029.287,E2 -16029.287} C_VEL
LIN {X 0,Y 305.454,Z 562.499,A -85,B 0,C 180,E1 -16030.942,E2 -16030.942} C_VEL
LIN {X 0,Y 306.153,Z 554.023,A -85,B 0,C 180,E1 -16032.26,E2 -16032.26} C_VEL
LIN {X 0,Y 306.73,Z 544.94,A -85,B 0,C 180,E1 -16033.414,E2 -16033.414} C_VEL
LIN {X 0,Y 307.119,Z 538.66,A -85,B 0,C 180,E1 -16034.072,E2 -16034.072} C_VEL
LIN {X 0,Y 305.727,Z 529.08,A -85,B 0,C 180,E1 -16034.944,E2 -16034.944} C_VEL
LIN {X 0,Y 304.012,Z 516.134,A -85,B 0,C 180,E1 -16035.858,E2 -16035.858} C_VEL
LIN {X 0,Y 304.062,Z 512.753,A -85,B 0,C 180,E1 -16038.88,E2 -16038.88} C_VEL
LIN {X 0,Y 304.242,Z 508.131,A -85,B 0,C 180,E1 -16043.123,E2 -16043.123} C_VEL
LIN {X 0,Y 304.278,Z 507.692,A -85,B 0,C 180,E1 -16043.57,E2 -16043.57} C_VEL
LIN {X 0,Y 305.578,Z 512.066,A -85,B 0,C 180,E1 -16046.237,E2 -16046.237} C_VEL
LIN {X 0,Y 305.921,Z 513.932,A -85,B 0,C 180,E1 -16047.353,E2 -16047.353} C_VEL
LIN {X 0,Y 305.531,Z 520.469,A -85,B 0,C 180,E1 -16051.026,E2 -16051.026} C_VEL
LIN {X 0,Y 305.182,Z 527.741,A -85,B 0,C 180,E1 -16055.15,E2 -16055.15} C_VEL
LIN {X 0,Y 305.087,Z 530.294,A -85,B 0,C 180,E1 -16056.478,E2 -16056.478} C_VEL
LIN {X 0,Y 307.549,Z 540.027,A -85,B 0,C 180,E1 -16057.167,E2 -16057.167} C_VEL
LIN {X 0,Y 309.314,Z 549.648,A -85,B 0,C 180,E1 -16057.992,E2 -16057.992} C_VEL
LIN {X 0,Y 310.479,Z 559.182,A -85,B 0,C 180,E1 -16058.977,E2 -16058.977} C_VEL
LIN {X 0,Y 309.963,Z 566.521,A -85,B 0,C 180,E1 -16059.818,E2 -16059.818} C_VEL
LIN {X 0,Y 308.833,Z 575.566,A -85,B 0,C 180,E1 -16061.077,E2 -16061.077} C_VEL
LIN {X 0,Y 307.767,Z 582.77,A -85,B 0,C 180,E1 -16062.327,E2 -16062.327} C_VEL
LIN {X 0,Y 306.71,Z 589.639,A -85,B 0,C 180,E1 -16063.796,E2 -16063.796} C_VEL
LIN {X 0,Y 305.775,Z 595.814,A -85,B 0,C 180,E1 -16065.44,E2 -16065.44} C_VEL
LIN {X 0,Y 304.924,Z 601.826,A -85,B 0,C 180,E1 -16067.523,E2 -16067.523} C_VEL
LIN {X 0,Y 304.441,Z 604.779,A -85,B 0,C 180,E1 -16068.859,E2 -16068.859} C_VEL
LIN {X 0,Y 304.023,Z 607.576,A -85,B 0,C 180,E1 -16070.527,E2 -16070.527} C_VEL
LIN {X 0,Y 303.726,Z 609.188,A -85,B 0,C 180,E1 -16071.882,E2 -16071.882} C_VEL
LIN {X 0,Y 303.454,Z 610.668,A -85,B 0,C 180,E1 -16074.155,E2 -16074.155} C_VEL
LIN {X 0,Y 303.344,Z 610.658,A -85,B 0,C 180,E1 -16076.519,E2 -16076.519} C_VEL
LIN {X 0,Y 303.526,Z 609.022,A -85,B 0,C 180,E1 -16078.95,E2 -16078.95} C_VEL
LIN {X 0,Y 303.864,Z 606.286,A -85,B 0,C 180,E1 -16080.941,E2 -16080.941} C_VEL
LIN {X 0,Y 304.114,Z 603.345,A -85,B 0,C 180,E1 -16082.47,E2 -16082.47} C_VEL
LIN {X 0,Y 304.529,Z 599.078,A -85,B 0,C 180,E1 -16084.165,E2 -16084.165} C_VEL
LIN {X 0,Y 305.163,Z 593.581,A -85,B 0,C 180,E1 -16085.871,E2 -16085.871} C_VEL
LIN {X 0,Y 306.005,Z 585.901,A -85,B 0,C 180,E1 -16087.73,E2 -16087.73} C_VEL
LIN {X 0,Y 306.823,Z 578.353,A -85,B 0,C 180,E1 -16089.148,E2 -16089.148} C_VEL
LIN {X 0,Y 307.62,Z 570.795,A -85,B 0,C 180,E1 -16090.306,E2 -16090.306} C_VEL
LIN {X 0,Y 308.283,Z 563.611,A -85,B 0,C 180,E1 -16091.215,E2 -16091.215} C_VEL
LIN {X 0,Y 308.668,Z 558.734,A -85,B 0,C 180,E1 -16091.755,E2 -16091.755} C_VEL
LIN {X 0,Y 307.491,Z 548.722,A -85,B 0,C 180,E1 -16092.714,E2 -16092.714} C_VEL
LIN {X 0,Y 306.017,Z 539.063,A -85,B 0,C 180,E1 -16093.445,E2 -16093.445} C_VEL
LIN {X 0,Y 304.349,Z 529.897,A -85,B 0,C 180,E1 -16093.998,E2 -16093.998} C_VEL
LIN {X 0,Y 304.634,Z 523.156,A -85,B 0,C 180,E1 -16098.016,E2 -16098.016} C_VEL
LIN {X 0,Y 304.962,Z 516.38,A -85,B 0,C 180,E1 -16102.051,E2 -16102.051} C_VEL
LIN {X 0,Y 305.258,Z 510.83,A -85,B 0,C 180,E1 -16105.377,E2 -16105.377} C_VEL
LIN {X 0,Y 305.395,Z 507.257,A -85,B 0,C 180,E1 -16107.609,E2 -16107.609} C_VEL
LIN {X 0,Y 305.964,Z 507.185,A -85,B 0,C 180,E1 -16109.999,E2 -16109.999} C_VEL
LIN {X 0,Y 305.888,Z 507.195,A -85,B 0,C 180,E1 -16112.633,E2 -16112.633} C_VEL
LIN {X 0,Y 305.854,Z 507.199,A -85,B 0,C 180,E1 -16116.597,E2 -16116.597} C_VEL
LIN {X 0,Y 305.737,Z 507.211,A -85,B 0,C 180,E1 -16119.259,E2 -16119.259} C_VEL
LIN {X 0,Y 305.589,Z 507.229,A -85,B 0,C 180,E1 -16123.295,E2 -16123.295} C_VEL
LIN {X 0,Y 305.594,Z 507.232,A -85,B 0,C 180,E1 -16126.019,E2 -16126.019} C_VEL
LIN {X 0,Y 305.577,Z 507.23,A -85,B 0,C 180,E1 -16129.444,E2 -16129.444} C_VEL
LIN {X 0,Y 305.49,Z 507.241,A -85,B 0,C 180,E1 -16133.041,E2 -16133.041} C_VEL
LIN {X 0,Y 305.548,Z 507.239,A -85,B 0,C 180,E1 -16136.227,E2 -16136.227} C_VEL
LIN {X 0,Y 305.503,Z 507.24,A -85,B 0,C 180,E1 -16139.052,E2 -16139.052} C_VEL
LIN {X 0,Y 305.464,Z 507.245,A -85,B 0,C 180,E1 -16143.516,E2 -16143.516} C_VEL
LIN {X 0,Y 305.494,Z 507.242,A -85,B 0,C 180,E1 -16146.736,E2 -16146.736} C_VEL
LIN {X 0,Y 305.457,Z 507.246,A -85,B 0,C 180,E1 -16150.6,E2 -16150.6} C_VEL
LIN {X 0,Y 305.483,Z 507.243,A -85,B 0,C 180,E1 -16153.644,E2 -16153.644} C_VEL
LIN {X 0,Y 305.507,Z 507.24,A -85,B 0,C 180,E1 -16157.402,E2 -16157.402} C_VEL
LIN {X 0,Y 305.518,Z 507.239,A -85,B 0,C 180,E1 -16161.604,E2 -16161.604} C_VEL
LIN {X 0,Y 305.46,Z 507.244,A -85,B 0,C 180,E1 -16164.886,E2 -16164.886} C_VEL
LIN {X 0,Y 305.449,Z 507.249,A -85,B 0,C 180,E1 -16168.354,E2 -16168.354} C_VEL
LIN {X 0,Y 305.517,Z 507.238,A -85,B 0,C 180,E1 -16171.113,E2 -16171.113} C_VEL
LIN {X 0,Y 305.569,Z 507.236,A -85,B 0,C 180,E1 -16174.088,E2 -16174.088} C_VEL
LIN {X 0,Y 305.498,Z 507.242,A -85,B 0,C 180,E1 -16178.403,E2 -16178.403} C_VEL
LIN {X 0,Y 305.588,Z 507.229,A -85,B 0,C 180,E1 -16181.217,E2 -16181.217} C_VEL
LIN {X 0,Y 305.646,Z 507.223,A -85,B 0,C 180,E1 -16185.349,E2 -16185.349} C_VEL
LIN {X 0,Y 305.591,Z 507.227,A -85,B 0,C 180,E1 -16186.174,E2 -16186.174} C_VEL
LIN {X 0,Y 304.932,Z 507.312,A -85,B 0,C 180,E1 -16187.273,E2 -16187.273} C_VEL
LIN {X 0,Y 302.175,Z 507.664,A -85,B 0,C 180,E1 -16189.066,E2 -16189.066} C_VEL
LIN {X 0,Y 299.842,Z 507.956,A -85,B 0,C 180,E1 -16190.52,E2 -16190.52} C_VEL
LIN {X 0,Y 298.837,Z 508.077,A -85,B 0,C 180,E1 -16191.644,E2 -16191.644} C_VEL
LIN {X 0,Y 298.753,Z 508.084,A -85,B 0,C 180,E1 -16192.025,E2 -16192.025} C_VEL
LIN {X 0,Y 298.658,Z 508.092,A -85,B 0,C 180,E1 -16194.599,E2 -16194.599} C_VEL
LIN {X 0,Y 298.923,Z 508.058,A -85,B 0,C 180,E1 -16198.653,E2 -16198.653} C_VEL
LIN {X 0,Y 298.921,Z 508.061,A -85,B 0,C 180,E1 -16201.347,E2 -16201.347} C_VEL
LIN {X 0,Y 298.795,Z 508.075,A -85,B 0,C 180,E1 -16206.754,E2 -16206.754} C_VEL
LIN {X 0,Y 298.678,Z 508.093,A -85,B 0,C 180,E1 -16209.48,E2 -16209.48} C_VEL
LIN {X 0,Y 298.549,Z 508.111,A -85,B 0,C 180,E1 -16213.615,E2 -16213.615} C_VEL
LIN {X 0,Y 298.546,Z 508.107,A -85,B 0,C 180,E1 -16216.409,E2 -16216.409} C_VEL
LIN {X 0,Y 298.508,Z 508.117,A -85,B 0,C 180,E1 -16219.655,E2 -16219.655} C_VEL
LIN {X 0,Y 298.454,Z 508.123,A -85,B 0,C 180,E1 -16223.598,E2 -16223.598} C_VEL
LIN {X 0,Y 298.486,Z 508.114,A -85,B 0,C 180,E1 -16226.575,E2 -16226.575} C_VEL
LIN {X 0,Y 298.419,Z 508.127,A -85,B 0,C 180,E1 -16229.641,E2 -16229.641} C_VEL
LIN {X 0,Y 298.395,Z 508.126,A -85,B 0,C 180,E1 -16232.8,E2 -16232.8} C_VEL
LIN {X 0,Y 298.462,Z 508.117,A -85,B 0,C 180,E1 -16236.813,E2 -16236.813} C_VEL
LIN {X 0,Y 298.409,Z 508.125,A -85,B 0,C 180,E1 -16241.094,E2 -16241.094} C_VEL
LIN {X 0,Y 298.423,Z 508.124,A -85,B 0,C 180,E1 -16243.109,E2 -16243.109} C_VEL
LIN {X 0,Y 298.429,Z 508.122,A -85,B 0,C 180,E1 -16246.926,E2 -16246.926} C_VEL
LIN {X 0,Y 298.578,Z 508.106,A -85,B 0,C 180,E1 -16251.84,E2 -16251.84} C_VEL
LIN {X 0,Y 298.638,Z 508.377,A -85,B 0,C 180,E1 -16252.276,E2 -16252.276} C_VEL
LIN {X 0,Y 299.786,Z 515.017,A -85,B 0,C 180,E1 -16256.571,E2 -16256.571} C_VEL
LIN {X 0,Y 299.976,Z 517.703,A -85,B 0,C 180,E1 -16258.247,E2 -16258.247} C_VEL
LIN {X 0,Y 299.059,Z 523.896,A -85,B 0,C 180,E1 -16261.966,E2 -16261.966} C_VEL
LIN {X 0,Y 298.125,Z 531.347,A -85,B 0,C 180,E1 -16266.375,E2 -16266.375} C_VEL
LIN {X 0,Y 297.377,Z 539.153,A -85,B 0,C 180,E1 -16270.967,E2 -16270.967} C_VEL
LIN {X 0,Y 297.255,Z 540.538,A -85,B 0,C 180,E1 -16271.759,E2 -16271.759} C_VEL
LIN {X 0,Y 298.786,Z 552.943,A -85,B 0,C 180,E1 -16272.328,E2 -16272.328} C_VEL
LIN {X 0,Y 299.663,Z 562.315,A -85,B 0,C 180,E1 -16272.953,E2 -16272.953} C_VEL
LIN {X 0,Y 300.214,Z 571.006,A -85,B 0,C 180,E1 -16273.701,E2 -16273.701} C_VEL
LIN {X 0,Y 300.53,Z 579.652,A -85,B 0,C 180,E1 -16274.629,E2 -16274.629} C_VEL
LIN {X 0,Y 300.034,Z 587.14,A -85,B 0,C 180,E1 -16275.589,E2 -16275.589} C_VEL
LIN {X 0,Y 299.192,Z 594.694,A -85,B 0,C 180,E1 -16276.761,E2 -16276.761} C_VEL
LIN {X 0,Y 298.267,Z 603.343,A -85,B 0,C 180,E1 -16278.447,E2 -16278.447} C_VEL
LIN {X 0,Y 297.579,Z 610.034,A -85,B 0,C 180,E1 -16280.142,E2 -16280.142} C_VEL
LIN {X 0,Y 297.072,Z 615.374,A -85,B 0,C 180,E1 -16281.84,E2 -16281.84} C_VEL
LIN {X 0,Y 296.768,Z 618.8,A -85,B 0,C 180,E1 -16283.2,E2 -16283.2} C_VEL
LIN {X 0,Y 296.639,Z 621.575,A -85,B 0,C 180,E1 -16284.563,E2 -16284.563} C_VEL
LIN {X 0,Y 296.625,Z 623.762,A -85,B 0,C 180,E1 -16285.925,E2 -16285.925} C_VEL
LIN {X 0,Y 296.582,Z 625.359,A -85,B 0,C 180,E1 -16287.284,E2 -16287.284} C_VEL
LIN {X 0,Y 296.534,Z 626.352,A -85,B 0,C 180,E1 -16288.643,E2 -16288.643} C_VEL
LIN {X 0,Y 296.574,Z 626.841,A -85,B 0,C 180,E1 -16290.001,E2 -16290.001} C_VEL
LIN {X 0,Y 296.531,Z 626.842,A -85,B 0,C 180,E1 -16291.359,E2 -16291.359} C_VEL
LIN {X 0,Y 296.575,Z 626.362,A -85,B 0,C 180,E1 -16292.717,E2 -16292.717} C_VEL
LIN {X 0,Y 296.593,Z 625.353,A -85,B 0,C 180,E1 -16294.077,E2 -16294.077} C_VEL
LIN {X 0,Y 296.679,Z 623.32,A -85,B 0,C 180,E1 -16295.772,E2 -16295.772} C_VEL
LIN {X 0,Y 297.658,Z 617.421,A -85,B 0,C 180,E1 -16299.514,E2 -16299.514} C_VEL
LIN {X 0,Y 298.717,Z 613.067,A -85,B 0,C 180,E1 -16301.537,E2 -16301.537} C_VEL
LIN {X 0,Y 300.226,Z 607.335,A -85,B 0,C 180,E1 -16303.539,E2 -16303.539} C_VEL
LIN {X 0,Y 302.108,Z 599.909,A -85,B 0,C 180,E1 -16305.518,E2 -16305.518} C_VEL
LIN {X 0,Y 303.592,Z 593.995,A -85,B 0,C 180,E1 -16306.821,E2 -16306.821} C_VEL
LIN {X 0,Y 305.164,Z 587.054,A -85,B 0,C 180,E1 -16308.115,E2 -16308.115} C_VEL
LIN {X 0,Y 306.115,Z 579.621,A -85,B 0,C 180,E1 -16309.351,E2 -16309.351} C_VEL
LIN {X 0,Y 306.169,Z 571.665,A -85,B 0,C 180,E1 -16310.619,E2 -16310.619} C_VEL
LIN {X 0,Y 305.196,Z 562.29,A -85,B 0,C 180,E1 -16312.05,E2 -16312.05} C_VEL
LIN {X 0,Y 303.195,Z 552.316,A -85,B 0,C 180,E1 -16313.57,E2 -16313.57} C_VEL
LIN {X 0,Y 300.787,Z 543.765,A -85,B 0,C 180,E1 -16314.872,E2 -16314.872} C_VEL
LIN {X 0,Y 299.594,Z 541.09,A -85,B 0,C 180,E1 -16315.349,E2 -16315.349} C_VEL
LIN {X 0,Y 299.141,Z 538.79,A -85,B 0,C 180,E1 -16315.67,E2 -16315.67} C_VEL
LIN {X 0,Y 300.236,Z 533.977,A -85,B 0,C 180,E1 -16319.445,E2 -16319.445} C_VEL
LIN {X 0,Y 301.201,Z 530.118,A -85,B 0,C 180,E1 -16322.861,E2 -16322.861} C_VEL
LIN {X 0,Y 301.529,Z 527.446,A -85,B 0,C 180,E1 -16325.641,E2 -16325.641} C_VEL
LIN {X 0,Y 301.48,Z 525.88,A -85,B 0,C 180,E1 -16327.571,E2 -16327.571} C_VEL
LIN {X 0,Y 301.174,Z 523.739,A -85,B 0,C 180,E1 -16330.798,E2 -16330.798} C_VEL
LIN {X 0,Y 300.894,Z 521.933,A -85,B 0,C 180,E1 -16334.485,E2 -16334.485} C_VEL
LIN {X 0,Y 300.677,Z 520.757,A -85,B 0,C 180,E1 -16338.415,E2 -16338.415} C_VEL
LIN {X 0,Y 300.539,Z 520.31,A -85,B 0,C 180,E1 -16342.555,E2 -16342.555} C_VEL
LIN {X 0,Y 300.361,Z 520.519,A -85,B 0,C 180,E1 -16345.836,E2 -16345.836} C_VEL
LIN {X 0,Y 300.04,Z 521.17,A -85,B 0,C 180,E1 -16348.981,E2 -16348.981} C_VEL
LIN {X 0,Y 299.51,Z 522.172,A -85,B 0,C 180,E1 -16352.011,E2 -16352.011} C_VEL
LIN {X 0,Y 299.159,Z 523.303,A -85,B 0,C 180,E1 -16354.519,E2 -16354.519} C_VEL
LIN {X 0,Y 300.406,Z 526.472,A -85,B 0,C 180,E1 -16355.095,E2 -16355.095} C_VEL
LIN {X 0,Y 301.842,Z 529.229,A -85,B 0,C 180,E1 -16355.709,E2 -16355.709} C_VEL
LIN {X 0,Y 305.492,Z 537.611,A -85,B 0,C 180,E1 -16357.394,E2 -16357.394} C_VEL
LIN {X 0,Y 308.318,Z 547.027,A -85,B 0,C 180,E1 -16359.162,E2 -16359.162} C_VEL
LIN {X 0,Y 309.61,Z 555.176,A -85,B 0,C 180,E1 -16360.679,E2 -16360.679} C_VEL
LIN {X 0,Y 307.725,Z 563.648,A -85,B 0,C 180,E1 -16362.042,E2 -16362.042} C_VEL
LIN {X 0,Y 306.093,Z 570.307,A -85,B 0,C 180,E1 -16363.321,E2 -16363.321} C_VEL
LIN {X 0,Y 304.142,Z 577.226,A -85,B 0,C 180,E1 -16364.932,E2 -16364.932} C_VEL
LIN {X 0,Y 302.474,Z 582.84,A -85,B 0,C 180,E1 -16366.565,E2 -16366.565} C_VEL
LIN {X 0,Y 300.73,Z 588.178,A -85,B 0,C 180,E1 -16368.542,E2 -16368.542} C_VEL
LIN {X 0,Y 299.425,Z 592.056,A -85,B 0,C 180,E1 -16370.543,E2 -16370.543} C_VEL
LIN {X 0,Y 298.491,Z 594.044,A -85,B 0,C 180,E1 -16371.879,E2 -16371.879} C_VEL
LIN {X 0,Y 297.999,Z 595.462,A -85,B 0,C 180,E1 -16373.228,E2 -16373.228} C_VEL
LIN {X 0,Y 297.72,Z 596.294,A -85,B 0,C 180,E1 -16374.582,E2 -16374.582} C_VEL
LIN {X 0,Y 297.325,Z 596.687,A -85,B 0,C 180,E1 -16375.934,E2 -16375.934} C_VEL
LIN {X 0,Y 296.999,Z 596.616,A -85,B 0,C 180,E1 -16377.287,E2 -16377.287} C_VEL
LIN {X 0,Y 296.758,Z 596.068,A -85,B 0,C 180,E1 -16378.643,E2 -16378.643} C_VEL
LIN {X 0,Y 296.661,Z 594.942,A -85,B 0,C 180,E1 -16380,E2 -16380} C_VEL
LIN {X 0,Y 296.658,Z 592.313,A -85,B 0,C 180,E1 -16382.037,E2 -16382.037} C_VEL
LIN {X 0,Y 296.848,Z 588.352,A -85,B 0,C 180,E1 -16384.073,E2 -16384.073} C_VEL
LIN {X 0,Y 296.95,Z 583.771,A -85,B 0,C 180,E1 -16385.845,E2 -16385.845} C_VEL
LIN {X 0,Y 297.376,Z 578.509,A -85,B 0,C 180,E1 -16387.469,E2 -16387.469} C_VEL
LIN {X 0,Y 297.718,Z 571.727,A -85,B 0,C 180,E1 -16389.169,E2 -16389.169} C_VEL
LIN {X 0,Y 298.326,Z 563.244,A -85,B 0,C 180,E1 -16390.863,E2 -16390.863} C_VEL
LIN {X 0,Y 298.979,Z 554.826,A -85,B 0,C 180,E1 -16392.214,E2 -16392.214} C_VEL
LIN {X 0,Y 299.592,Z 545.857,A -85,B 0,C 180,E1 -16393.395,E2 -16393.395} C_VEL
LIN {X 0,Y 299.932,Z 538.02,A -85,B 0,C 180,E1 -16394.243,E2 -16394.243} C_VEL
LIN {X 0,Y 298.312,Z 527.148,A -85,B 0,C 180,E1 -16395.228,E2 -16395.228} C_VEL
LIN {X 0,Y 296.938,Z 516.477,A -85,B 0,C 180,E1 -16395.97,E2 -16395.97} C_VEL
LIN {X 0,Y 296.967,Z 512.766,A -85,B 0,C 180,E1 -16399.349,E2 -16399.349} C_VEL
LIN {X 0,Y 297.174,Z 508.676,A -85,B 0,C 180,E1 -16403.208,E2 -16403.208} C_VEL
LIN {X 0,Y 298.468,Z 512.84,A -85,B 0,C 180,E1 -16405.825,E2 -16405.825} C_VEL
LIN {X 0,Y 298.947,Z 515.233,A -85,B 0,C 180,E1 -16407.285,E2 -16407.285} C_VEL
LIN {X 0,Y 298.618,Z 520.658,A -85,B 0,C 180,E1 -16410.398,E2 -16410.398} C_VEL
LIN {X 0,Y 298.218,Z 527.721,A -85,B 0,C 180,E1 -16414.444,E2 -16414.444} C_VEL
LIN {X 0,Y 298.123,Z 530.434,A -85,B 0,C 180,E1 -16415.903,E2 -16415.903} C_VEL
LIN {X 0,Y 300.672,Z 540.409,A -85,B 0,C 180,E1 -16416.645,E2 -16416.645} C_VEL
LIN {X 0,Y 302.326,Z 549.113,A -85,B 0,C 180,E1 -16417.417,E2 -16417.417} C_VEL
LIN {X 0,Y 303.51,Z 557.528,A -85,B 0,C 180,E1 -16418.302,E2 -16418.302} C_VEL
LIN {X 0,Y 303.706,Z 563.063,A -85,B 0,C 180,E1 -16418.948,E2 -16418.948} C_VEL
LIN {X 0,Y 302.675,Z 571.198,A -85,B 0,C 180,E1 -16419.981,E2 -16419.981} C_VEL
LIN {X 0,Y 301.5,Z 579.588,A -85,B 0,C 180,E1 -16421.305,E2 -16421.305} C_VEL
LIN {X 0,Y 300.097,Z 588.307,A -85,B 0,C 180,E1 -16423.06,E2 -16423.06} C_VEL
LIN {X 0,Y 299.178,Z 594.151,A -85,B 0,C 180,E1 -16424.566,E2 -16424.566} C_VEL
LIN {X 0,Y 298.43,Z 598.692,A -85,B 0,C 180,E1 -16425.994,E2 -16425.994} C_VEL
LIN {X 0,Y 297.731,Z 603.169,A -85,B 0,C 180,E1 -16427.777,E2 -16427.777} C_VEL
LIN {X 0,Y 297.274,Z 605.894,A -85,B 0,C 180,E1 -16429.159,E2 -16429.159} C_VEL
LIN {X 0,Y 296.984,Z 607.715,A -85,B 0,C 180,E1 -16430.286,E2 -16430.286} C_VEL
LIN {X 0,Y 296.632,Z 609.641,A -85,B 0,C 180,E1 -16431.974,E2 -16431.974} C_VEL
LIN {X 0,Y 296.398,Z 610.788,A -85,B 0,C 180,E1 -16433.725,E2 -16433.725} C_VEL
LIN {X 0,Y 296.268,Z 611.111,A -85,B 0,C 180,E1 -16435.296,E2 -16435.296} C_VEL
LIN {X 0,Y 296.257,Z 610.725,A -85,B 0,C 180,E1 -16436.932,E2 -16436.932} C_VEL
LIN {X 0,Y 296.38,Z 609.565,A -85,B 0,C 180,E1 -16438.612,E2 -16438.612} C_VEL
LIN {X 0,Y 296.64,Z 607.77,A -85,B 0,C 180,E1 -16440.162,E2 -16440.162} C_VEL
LIN {X 0,Y 296.902,Z 605.206,A -85,B 0,C 180,E1 -16441.743,E2 -16441.743} C_VEL
LIN {X 0,Y 297.375,Z 600.335,A -85,B 0,C 180,E1 -16443.906,E2 -16443.906} C_VEL
LIN {X 0,Y 297.98,Z 595.179,A -85,B 0,C 180,E1 -16445.622,E2 -16445.622} C_VEL
LIN {X 0,Y 298.632,Z 589.405,A -85,B 0,C 180,E1 -16447.164,E2 -16447.164} C_VEL
LIN {X 0,Y 299.402,Z 582.496,A -85,B 0,C 180,E1 -16448.663,E2 -16448.663} C_VEL
LIN {X 0,Y 300.38,Z 573.832,A -85,B 0,C 180,E1 -16450.168,E2 -16450.168} C_VEL
LIN {X 0,Y 301.174,Z 565.655,A -85,B 0,C 180,E1 -16451.284,E2 -16451.284} C_VEL
LIN {X 0,Y 301.697,Z 559.249,A -85,B 0,C 180,E1 -16452.021,E2 -16452.021} C_VEL
LIN {X 0,Y 300.534,Z 549.357,A -85,B 0,C 180,E1 -16453.003,E2 -16453.003} C_VEL
LIN {X 0,Y 299.105,Z 539.8,A -85,B 0,C 180,E1 -16453.754,E2 -16453.754} C_VEL
LIN {X 0,Y 297.338,Z 530.033,A -85,B 0,C 180,E1 -16454.359,E2 -16454.359} C_VEL
LIN {X 0,Y 297.634,Z 523.322,A -85,B 0,C 180,E1 -16458.421,E2 -16458.421} C_VEL
LIN {X 0,Y 297.945,Z 517.086,A -85,B 0,C 180,E1 -16462.183,E2 -16462.183} C_VEL
LIN {X 0,Y 298.219,Z 510.929,A -85,B 0,C 180,E1 -16465.945,E2 -16465.945} C_VEL
LIN {X 0,Y 298.368,Z 508.132,A -85,B 0,C 180,E1 -16467.637,E2 -16467.637} C_VEL
LIN {X 0,Y 298.921,Z 508.063,A -85,B 0,C 180,E1 -16469.999,E2 -16469.999} C_VEL
LIN {X 0,Y 298.839,Z 508.073,A -85,B 0,C 180,E1 -16472.695,E2 -16472.695} C_VEL
LIN {X 0,Y 298.799,Z 508.077,A -85,B 0,C 180,E1 -16476.753,E2 -16476.753} C_VEL
LIN {X 0,Y 298.681,Z 508.09,A -85,B 0,C 180,E1 -16479.48,E2 -16479.48} C_VEL
LIN {X 0,Y 298.553,Z 508.106,A -85,B 0,C 180,E1 -16483.615,E2 -16483.615} C_VEL
LIN {X 0,Y 298.549,Z 508.11,A -85,B 0,C 180,E1 -16486.408,E2 -16486.408} C_VEL
LIN {X 0,Y 298.512,Z 508.111,A -85,B 0,C 180,E1 -16489.654,E2 -16489.654} C_VEL
LIN {X 0,Y 298.457,Z 508.118,A -85,B 0,C 180,E1 -16493.597,E2 -16493.597} C_VEL
LIN {X 0,Y 298.49,Z 508.115,A -85,B 0,C 180,E1 -16496.574,E2 -16496.574} C_VEL
LIN {X 0,Y 298.424,Z 508.123,A -85,B 0,C 180,E1 -16499.64,E2 -16499.64} C_VEL
LIN {X 0,Y 298.395,Z 508.126,A -85,B 0,C 180,E1 -16502.799,E2 -16502.799} C_VEL
LIN {X 0,Y 298.463,Z 508.117,A -85,B 0,C 180,E1 -16506.812,E2 -16506.812} C_VEL
LIN {X 0,Y 298.415,Z 508.122,A -85,B 0,C 180,E1 -16511.255,E2 -16511.255} C_VEL
LIN {X 0,Y 298.415,Z 508.122,A -85,B 0,C 180,E1 -16514.953,E2 -16514.953} C_VEL
LIN {X 0,Y 298.453,Z 508.118,A -85,B 0,C 180,E1 -16518.75,E2 -16518.75} C_VEL
LIN {X 0,Y 298.445,Z 508.121,A -85,B 0,C 180,E1 -16522.246,E2 -16522.246} C_VEL
LIN {X 0,Y 298.406,Z 508.125,A -85,B 0,C 180,E1 -16525.581,E2 -16525.581} C_VEL
LIN {X 0,Y 298.392,Z 508.126,A -85,B 0,C 180,E1 -16528.791,E2 -16528.791} C_VEL
LIN {X 0,Y 298.46,Z 508.122,A -85,B 0,C 180,E1 -16531.904,E2 -16531.904} C_VEL
LIN {X 0,Y 298.483,Z 508.114,A -85,B 0,C 180,E1 -16534.924,E2 -16534.924} C_VEL
LIN {X 0,Y 298.447,Z 508.119,A -85,B 0,C 180,E1 -16539.315,E2 -16539.315} C_VEL
LIN {X 0,Y 298.535,Z 508.11,A -85,B 0,C 180,E1 -16542.179,E2 -16542.179} C_VEL
LIN {X 0,Y 298.591,Z 508.101,A -85,B 0,C 180,E1 -16544.995,E2 -16544.995} C_VEL
LIN {X 0,Y 298.593,Z 508.1,A -85,B 0,C 180,E1 -16549.147,E2 -16549.147} C_VEL
LIN {X 0,Y 298.753,Z 508.084,A -85,B 0,C 180,E1 -16552.025,E2 -16552.025} C_VEL
LIN {X 0,Y 298.073,Z 508.167,A -85,B 0,C 180,E1 -16553.148,E2 -16553.148} C_VEL
LIN {X 0,Y 295.221,Z 508.521,A -85,B 0,C 180,E1 -16554.979,E2 -16554.979} C_VEL
LIN {X 0,Y 292.844,Z 508.816,A -85,B 0,C 180,E1 -16556.464,E2 -16556.464} C_VEL
LIN {X 0,Y 291.875,Z 508.94,A -85,B 0,C 180,E1 -16557.615,E2 -16557.615} C_VEL
LIN {X 0,Y 291.823,Z 508.94,A -85,B 0,C 180,E1 -16558.004,E2 -16558.004} C_VEL
LIN {X 0,Y 291.964,Z 508.929,A -85,B 0,C 180,E1 -16560,E2 -16560} C_VEL
LIN {X 0,Y 291.789,Z 508.948,A -85,B 0,C 180,E1 -16562.761,E2 -16562.761} C_VEL
LIN {X 0,Y 291.744,Z 508.954,A -85,B 0,C 180,E1 -16566.918,E2 -16566.918} C_VEL
LIN {X 0,Y 291.626,Z 508.974,A -85,B 0,C 180,E1 -16569.712,E2 -16569.712} C_VEL
LIN {X 0,Y 291.519,Z 508.985,A -85,B 0,C 180,E1 -16573.95,E2 -16573.95} C_VEL
LIN {X 0,Y 291.484,Z 508.986,A -85,B 0,C 180,E1 -16576.818,E2 -16576.818} C_VEL
LIN {X 0,Y 291.447,Z 508.994,A -85,B 0,C 180,E1 -16579.875,E2 -16579.875} C_VEL
LIN {X 0,Y 291.397,Z 508.998,A -85,B 0,C 180,E1 -16584.205,E2 -16584.205} C_VEL
LIN {X 0,Y 291.42,Z 508.997,A -85,B 0,C 180,E1 -16587.272,E2 -16587.272} C_VEL
LIN {X 0,Y 291.337,Z 509.005,A -85,B 0,C 180,E1 -16590.437,E2 -16590.437} C_VEL
LIN {X 0,Y 291.343,Z 509.008,A -85,B 0,C 180,E1 -16593.698,E2 -16593.698} C_VEL
LIN {X 0,Y 291.392,Z 509,A -85,B 0,C 180,E1 -16597.259,E2 -16597.259} C_VEL
LIN {X 0,Y 291.348,Z 509.003,A -85,B 0,C 180,E1 -16600.64,E2 -16600.64} C_VEL
LIN {X 0,Y 291.32,Z 509.007,A -85,B 0,C 180,E1 -16604.396,E2 -16604.396} C_VEL
LIN {X 0,Y 291.349,Z 509.008,A -85,B 0,C 180,E1 -16607.514,E2 -16607.514} C_VEL
LIN {X 0,Y 291.582,Z 509.131,A -85,B 0,C 180,E1 -16612.186,E2 -16612.186} C_VEL
LIN {X 0,Y 292.703,Z 515.605,A -85,B 0,C 180,E1 -16616.48,E2 -16616.48} C_VEL
LIN {X 0,Y 292.9,Z 518.191,A -85,B 0,C 180,E1 -16618.139,E2 -16618.139} C_VEL
LIN {X 0,Y 291.966,Z 524.46,A -85,B 0,C 180,E1 -16622.006,E2 -16622.006} C_VEL
LIN {X 0,Y 291.132,Z 530.641,A -85,B 0,C 180,E1 -16625.772,E2 -16625.772} C_VEL
LIN {X 0,Y 290.389,Z 537.942,A -85,B 0,C 180,E1 -16630.195,E2 -16630.195} C_VEL
LIN {X 0,Y 290.218,Z 539.842,A -85,B 0,C 180,E1 -16631.344,E2 -16631.344} C_VEL
LIN {X 0,Y 291.816,Z 553.017,A -85,B 0,C 180,E1 -16631.982,E2 -16631.982} C_VEL
LIN {X 0,Y 292.675,Z 562.311,A -85,B 0,C 180,E1 -16632.624,E2 -16632.624} C_VEL
LIN {X 0,Y 293.173,Z 569.872,A -85,B 0,C 180,E1 -16633.282,E2 -16633.282} C_VEL
LIN {X 0,Y 293.515,Z 578.123,A -85,B 0,C 180,E1 -16634.168,E2 -16634.168} C_VEL
LIN {X 0,Y 293.227,Z 585.222,A -85,B 0,C 180,E1 -16635.07,E2 -16635.07} C_VEL
LIN {X 0,Y 292.341,Z 593.063,A -85,B 0,C 180,E1 -16636.268,E2 -16636.268} C_VEL
LIN {X 0,Y 291.621,Z 599.537,A -85,B 0,C 180,E1 -16637.474,E2 -16637.474} C_VEL
LIN {X 0,Y 290.94,Z 605.681,A -85,B 0,C 180,E1 -16638.858,E2 -16638.858} C_VEL
LIN {X 0,Y 290.332,Z 611.941,A -85,B 0,C 180,E1 -16640.597,E2 -16640.597} C_VEL
LIN {X 0,Y 289.851,Z 616.882,A -85,B 0,C 180,E1 -16642.337,E2 -16642.337} C_VEL
LIN {X 0,Y 289.555,Z 621.263,A -85,B 0,C 180,E1 -16644.429,E2 -16644.429} C_VEL
LIN {X 0,Y 289.519,Z 623.484,A -85,B 0,C 180,E1 -16645.825,E2 -16645.825} C_VEL
LIN {X 0,Y 289.509,Z 625.093,A -85,B 0,C 180,E1 -16647.218,E2 -16647.218} C_VEL
LIN {X 0,Y 289.454,Z 626.111,A -85,B 0,C 180,E1 -16648.609,E2 -16648.609} C_VEL
LIN {X 0,Y 289.488,Z 626.633,A -85,B 0,C 180,E1 -16650.001,E2 -16650.001} C_VEL
LIN {X 0,Y 289.451,Z 626.667,A -85,B 0,C 180,E1 -16651.392,E2 -16651.392} C_VEL
LIN {X 0,Y 289.501,Z 626.219,A -85,B 0,C 180,E1 -16652.784,E2 -16652.784} C_VEL
LIN {X 0,Y 289.498,Z 625.218,A -85,B 0,C 180,E1 -16654.177,E2 -16654.177} C_VEL
LIN {X 0,Y 289.593,Z 623.45,A -85,B 0,C 180,E1 -16655.728,E2 -16655.728} C_VEL
LIN {X 0,Y 290.651,Z 617.605,A -85,B 0,C 180,E1 -16659.746,E2 -16659.746} C_VEL
LIN {X 0,Y 291.772,Z 613.417,A -85,B 0,C 180,E1 -16661.815,E2 -16661.815} C_VEL
LIN {X 0,Y 293.377,Z 607.982,A -85,B 0,C 180,E1 -16663.861,E2 -16663.861} C_VEL
LIN {X 0,Y 295.355,Z 600.99,A -85,B 0,C 180,E1 -16665.882,E2 -16665.882} C_VEL
LIN {X 0,Y 296.904,Z 595.332,A -85,B 0,C 180,E1 -16667.211,E2 -16667.211} C_VEL
LIN {X 0,Y 298.619,Z 588.721,A -85,B 0,C 180,E1 -16668.526,E2 -16668.526} C_VEL
LIN {X 0,Y 299.823,Z 580.524,A -85,B 0,C 180,E1 -16669.993,E2 -16669.993} C_VEL
LIN {X 0,Y 299.959,Z 572.781,A -85,B 0,C 180,E1 -16671.295,E2 -16671.295} C_VEL
LIN {X 0,Y 299.016,Z 563.096,A -85,B 0,C 180,E1 -16672.899,E2 -16672.899} C_VEL
LIN {X 0,Y 296.808,Z 552.053,A -85,B 0,C 180,E1 -16674.725,E2 -16674.725} C_VEL
LIN {X 0,Y 294.02,Z 542.841,A -85,B 0,C 180,E1 -16676.317,E2 -16676.317} C_VEL
LIN {X 0,Y 292.643,Z 538.775,A -85,B 0,C 180,E1 -16677.035,E2 -16677.035} C_VEL
LIN {X 0,Y 292.572,Z 538.091,A -85,B 0,C 180,E1 -16677.156,E2 -16677.156} C_VEL
LIN {X 0,Y 293.52,Z 534.152,A -85,B 0,C 180,E1 -16680.461,E2 -16680.461} C_VEL
LIN {X 0,Y 294.317,Z 531.103,A -85,B 0,C 180,E1 -16683.314,E2 -16683.314} C_VEL
LIN {X 0,Y 294.587,Z 528.835,A -85,B 0,C 180,E1 -16685.793,E2 -16685.793} C_VEL
LIN {X 0,Y 294.457,Z 526.886,A -85,B 0,C 180,E1 -16688.358,E2 -16688.358} C_VEL
LIN {X 0,Y 294.149,Z 524.582,A -85,B 0,C 180,E1 -16692.211,E2 -16692.211} C_VEL
LIN {X 0,Y 293.903,Z 522.993,A -85,B 0,C 180,E1 -16696.095,E2 -16696.095} C_VEL
LIN {X 0,Y 293.7,Z 522.123,A -85,B 0,C 180,E1 -16699.973,E2 -16699.973} C_VEL
LIN {X 0,Y 293.586,Z 521.914,A -85,B 0,C 180,E1 -16703.24,E2 -16703.24} C_VEL
LIN {X 0,Y 293.357,Z 522.192,A -85,B 0,C 180,E1 -16706.564,E2 -16706.564} C_VEL
LIN {X 0,Y 292.97,Z 522.897,A -85,B 0,C 180,E1 -16709.751,E2 -16709.751} C_VEL
LIN {X 0,Y 292.435,Z 524.012,A -85,B 0,C 180,E1 -16712.996,E2 -16712.996} C_VEL
LIN {X 0,Y 292.841,Z 525.514,A -85,B 0,C 180,E1 -16713.257,E2 -16713.257} C_VEL
LIN {X 0,Y 294.799,Z 528.974,A -85,B 0,C 180,E1 -16714.153,E2 -16714.153} C_VEL
LIN {X 0,Y 299.154,Z 538.927,A -85,B 0,C 180,E1 -16716.382,E2 -16716.382} C_VEL
LIN {X 0,Y 301.831,Z 547.396,A -85,B 0,C 180,E1 -16718.127,E2 -16718.127} C_VEL
LIN {X 0,Y 303.206,Z 555.013,A -85,B 0,C 180,E1 -16719.654,E2 -16719.654} C_VEL
LIN {X 0,Y 303.409,Z 556.779,A -85,B 0,C 180,E1 -16720.022,E2 -16720.022} C_VEL
LIN {X 0,Y 302.744,Z 560.73,A -85,B 0,C 180,E1 -16720.683,E2 -16720.683} C_VEL
LIN {X 0,Y 300.404,Z 569.464,A -85,B 0,C 180,E1 -16722.294,E2 -16722.294} C_VEL
LIN {X 0,Y 298.251,Z 576.518,A -85,B 0,C 180,E1 -16723.926,E2 -16723.926} C_VEL
LIN {X 0,Y 296.397,Z 582.337,A -85,B 0,C 180,E1 -16725.584,E2 -16725.584} C_VEL
LIN {X 0,Y 294.468,Z 587.904,A -85,B 0,C 180,E1 -16727.596,E2 -16727.596} C_VEL
LIN {X 0,Y 293.141,Z 591.609,A -85,B 0,C 180,E1 -16729.413,E2 -16729.413} C_VEL
LIN {X 0,Y 291.522,Z 594.843,A -85,B 0,C 180,E1 -16731.683,E2 -16731.683} C_VEL
LIN {X 0,Y 290.98,Z 596.148,A -85,B 0,C 180,E1 -16733.064,E2 -16733.064} C_VEL
LIN {X 0,Y 290.67,Z 596.923,A -85,B 0,C 180,E1 -16734.45,E2 -16734.45} C_VEL
LIN {X 0,Y 290.258,Z 597.152,A -85,B 0,C 180,E1 -16735.835,E2 -16735.835} C_VEL
LIN {X 0,Y 289.919,Z 596.92,A -85,B 0,C 180,E1 -16737.221,E2 -16737.221} C_VEL
LIN {X 0,Y 289.673,Z 596.229,A -85,B 0,C 180,E1 -16738.61,E2 -16738.61} C_VEL
LIN {X 0,Y 289.573,Z 595.044,A -85,B 0,C 180,E1 -16740,E2 -16740} C_VEL
LIN {X 0,Y 289.58,Z 592.157,A -85,B 0,C 180,E1 -16742.086,E2 -16742.086} C_VEL
LIN {X 0,Y 289.721,Z 589.608,A -85,B 0,C 180,E1 -16743.477,E2 -16743.477} C_VEL
LIN {X 0,Y 289.852,Z 584.482,A -85,B 0,C 180,E1 -16745.566,E2 -16745.566} C_VEL
LIN {X 0,Y 290.198,Z 579.06,A -85,B 0,C 180,E1 -16747.305,E2 -16747.305} C_VEL
LIN {X 0,Y 290.529,Z 573.794,A -85,B 0,C 180,E1 -16748.696,E2 -16748.696} C_VEL
LIN {X 0,Y 290.939,Z 567.513,A -85,B 0,C 180,E1 -16750.086,E2 -16750.086} C_VEL
LIN {X 0,Y 291.6,Z 559.003,A -85,B 0,C 180,E1 -16751.645,E2 -16751.645} C_VEL
LIN {X 0,Y 292.221,Z 549.532,A -85,B 0,C 180,E1 -16753.031,E2 -16753.031} C_VEL
LIN {X 0,Y 292.89,Z 539.5,A -85,B 0,C 180,E1 -16754.194,E2 -16754.194} C_VEL
LIN {X 0,Y 291.415,Z 529.14,A -85,B 0,C 180,E1 -16755.182,E2 -16755.182} C_VEL
LIN {X 0,Y 289.858,Z 516.794,A -85,B 0,C 180,E1 -16756.1,E2 -16756.1} C_VEL
LIN {X 0,Y 289.901,Z 512.76,A -85,B 0,C 180,E1 -16759.84,E2 -16759.84} C_VEL
LIN {X 0,Y 290.082,Z 509.652,A -85,B 0,C 180,E1 -16762.808,E2 -16762.808} C_VEL
LIN {X 0,Y 291.495,Z 514.189,A -85,B 0,C 180,E1 -16765.721,E2 -16765.721} C_VEL
LIN {X 0,Y 292,Z 516.59,A -85,B 0,C 180,E1 -16767.213,E2 -16767.213} C_VEL
LIN {X 0,Y 291.541,Z 523.417,A -85,B 0,C 180,E1 -16771.218,E2 -16771.218} C_VEL
LIN {X 0,Y 291.161,Z 530.354,A -85,B 0,C 180,E1 -16775.261,E2 -16775.261} C_VEL
LIN {X 0,Y 294.154,Z 542.113,A -85,B 0,C 180,E1 -16776.199,E2 -16776.199} C_VEL
LIN {X 0,Y 296.159,Z 553.439,A -85,B 0,C 180,E1 -16777.297,E2 -16777.297} C_VEL
LIN {X 0,Y 297.048,Z 562.191,A -85,B 0,C 180,E1 -16778.336,E2 -16778.336} C_VEL
LIN {X 0,Y 296.15,Z 570.067,A -85,B 0,C 180,E1 -16779.336,E2 -16779.336} C_VEL
LIN {X 0,Y 295.022,Z 578.128,A -85,B 0,C 180,E1 -16780.595,E2 -16780.595} C_VEL
LIN {X 0,Y 294.049,Z 583.914,A -85,B 0,C 180,E1 -16781.677,E2 -16781.677} C_VEL
LIN {X 0,Y 293.037,Z 589.767,A -85,B 0,C 180,E1 -16782.988,E2 -16782.988} C_VEL
LIN {X 0,Y 292.064,Z 595.501,A -85,B 0,C 180,E1 -16784.56,E2 -16784.56} C_VEL
LIN {X 0,Y 291.309,Z 599.957,A -85,B 0,C 180,E1 -16786.071,E2 -16786.071} C_VEL
LIN {X 0,Y 290.782,Z 603.179,A -85,B 0,C 180,E1 -16787.41,E2 -16787.41} C_VEL
LIN {X 0,Y 290.188,Z 606.493,A -85,B 0,C 180,E1 -16789.162,E2 -16789.162} C_VEL
LIN {X 0,Y 289.734,Z 608.887,A -85,B 0,C 180,E1 -16790.915,E2 -16790.915} C_VEL
LIN {X 0,Y 289.339,Z 610.834,A -85,B 0,C 180,E1 -16793.28,E2 -16793.28} C_VEL
LIN {X 0,Y 289.163,Z 611.138,A -85,B 0,C 180,E1 -16796.012,E2 -16796.012} C_VEL
LIN {X 0,Y 289.262,Z 610.008,A -85,B 0,C 180,E1 -16798.252,E2 -16798.252} C_VEL
LIN {X 0,Y 289.557,Z 607.995,A -85,B 0,C 180,E1 -16800.16,E2 -16800.16} C_VEL
LIN {X 0,Y 289.812,Z 605.447,A -85,B 0,C 180,E1 -16801.778,E2 -16801.778} C_VEL
LIN {X 0,Y 290.23,Z 601.554,A -85,B 0,C 180,E1 -16803.633,E2 -16803.633} C_VEL
LIN {X 0,Y 290.748,Z 596.791,A -85,B 0,C 180,E1 -16805.356,E2 -16805.356} C_VEL
LIN {X 0,Y 291.397,Z 591.371,A -85,B 0,C 180,E1 -16806.92,E2 -16806.92} C_VEL
LIN {X 0,Y 292.173,Z 584.694,A -85,B 0,C 180,E1 -16808.479,E2 -16808.479} C_VEL
LIN {X 0,Y 292.971,Z 577.877,A -85,B 0,C 180,E1 -16809.782,E2 -16809.782} C_VEL
LIN {X 0,Y 293.835,Z 570.237,A -85,B 0,C 180,E1 -16810.98,E2 -16810.98} C_VEL
LIN {X 0,Y 294.723,Z 559.745,A -85,B 0,C 180,E1 -16812.299,E2 -16812.299} C_VEL
LIN {X 0,Y 293.571,Z 549.947,A -85,B 0,C 180,E1 -16813.304,E2 -16813.304} C_VEL
LIN {X 0,Y 292.07,Z 539.966,A -85,B 0,C 180,E1 -16814.109,E2 -16814.109} C_VEL
LIN {X 0,Y 290.301,Z 530.191,A -85,B 0,C 180,E1 -16814.718,E2 -16814.718} C_VEL
LIN {X 0,Y 290.614,Z 523.47,A -85,B 0,C 180,E1 -16818.844,E2 -16818.844} C_VEL
LIN {X 0,Y 290.94,Z 516.611,A -85,B 0,C 180,E1 -16823.062,E2 -16823.062} C_VEL
LIN {X 0,Y 291.238,Z 510.943,A -85,B 0,C 180,E1 -16826.541,E2 -16826.541} C_VEL
LIN {X 0,Y 291.359,Z 509.006,A -85,B 0,C 180,E1 -16827.753,E2 -16827.753} C_VEL
LIN {X 0,Y 291.879,Z 508.94,A -85,B 0,C 180,E1 -16829.999,E2 -16829.999} C_VEL
LIN {X 0,Y 291.791,Z 508.95,A -85,B 0,C 180,E1 -16832.76,E2 -16832.76} C_VEL
LIN {X 0,Y 291.748,Z 508.954,A -85,B 0,C 180,E1 -16836.917,E2 -16836.917} C_VEL
LIN {X 0,Y 291.63,Z 508.969,A -85,B 0,C 180,E1 -16839.711,E2 -16839.711} C_VEL
LIN {X 0,Y 291.522,Z 508.984,A -85,B 0,C 180,E1 -16843.949,E2 -16843.949} C_VEL
LIN {X 0,Y 291.487,Z 508.987,A -85,B 0,C 180,E1 -16846.817,E2 -16846.817} C_VEL
LIN {X 0,Y 291.451,Z 508.992,A -85,B 0,C 180,E1 -16849.874,E2 -16849.874} C_VEL
LIN {X 0,Y 291.4,Z 509.001,A -85,B 0,C 180,E1 -16854.204,E2 -16854.204} C_VEL
LIN {X 0,Y 291.425,Z 508.993,A -85,B 0,C 180,E1 -16857.27,E2 -16857.27} C_VEL
LIN {X 0,Y 291.338,Z 509.007,A -85,B 0,C 180,E1 -16860.436,E2 -16860.436} C_VEL
LIN {X 0,Y 291.344,Z 509.005,A -85,B 0,C 180,E1 -16863.698,E2 -16863.698} C_VEL
LIN {X 0,Y 291.392,Z 508.997,A -85,B 0,C 180,E1 -16867.258,E2 -16867.258} C_VEL
LIN {X 0,Y 291.372,Z 509.001,A -85,B 0,C 180,E1 -16870.635,E2 -16870.635} C_VEL
LIN {X 0,Y 291.351,Z 509.005,A -85,B 0,C 180,E1 -16874.389,E2 -16874.389} C_VEL
LIN {X 0,Y 291.387,Z 509,A -85,B 0,C 180,E1 -16878.39,E2 -16878.39} C_VEL
LIN {X 0,Y 291.386,Z 508.998,A -85,B 0,C 180,E1 -16881.163,E2 -16881.163} C_VEL
LIN {X 0,Y 291.384,Z 508.998,A -85,B 0,C 180,E1 -16884.629,E2 -16884.629} C_VEL
LIN {X 0,Y 291.37,Z 509.005,A -85,B 0,C 180,E1 -16887.95,E2 -16887.95} C_VEL
LIN {X 0,Y 291.379,Z 508.999,A -85,B 0,C 180,E1 -16891.158,E2 -16891.158} C_VEL
LIN {X 0,Y 291.414,Z 508.997,A -85,B 0,C 180,E1 -16894.272,E2 -16894.272} C_VEL
LIN {X 0,Y 291.379,Z 509,A -85,B 0,C 180,E1 -16897.299,E2 -16897.299} C_VEL
LIN {X 0,Y 291.455,Z 508.991,A -85,B 0,C 180,E1 -16900.27,E2 -16900.27} C_VEL
LIN {X 0,Y 291.552,Z 508.978,A -85,B 0,C 180,E1 -16904.623,E2 -16904.623} C_VEL
LIN {X 0,Y 291.536,Z 508.979,A -85,B 0,C 180,E1 -16908.88,E2 -16908.88} C_VEL
LIN {X 0,Y 291.7,Z 508.96,A -85,B 0,C 180,E1 -16912.023,E2 -16912.023} C_VEL
LIN {X 0,Y 291.629,Z 508.968,A -85,B 0,C 180,E1 -16914.468,E2 -16914.468} C_VEL
LIN {X 0,Y 291.823,Z 508.94,A -85,B 0,C 180,E1 -16918.004,E2 -16918.004} C_VEL
LIN {X 0,Y 291.217,Z 509.019,A -85,B 0,C 180,E1 -16919.156,E2 -16919.156} C_VEL
LIN {X 0,Y 288.335,Z 509.378,A -85,B 0,C 180,E1 -16921.031,E2 -16921.031} C_VEL
LIN {X 0,Y 285.801,Z 509.694,A -85,B 0,C 180,E1 -16922.553,E2 -16922.553} C_VEL
LIN {X 0,Y 284.648,Z 509.843,A -85,B 0,C 180,E1 -16923.733,E2 -16923.733} C_VEL
LIN {X 0,Y 284.522,Z 509.854,A -85,B 0,C 180,E1 -16924.135,E2 -16924.135} C_VEL
LIN {X 0,Y 284.696,Z 509.832,A -85,B 0,C 180,E1 -16927.09,E2 -16927.09} C_VEL
LIN {X 0,Y 284.564,Z 509.851,A -85,B 0,C 180,E1 -16929.955,E2 -16929.955} C_VEL
LIN {X 0,Y 284.479,Z 509.86,A -85,B 0,C 180,E1 -16934.303,E2 -16934.303} C_VEL
LIN {X 0,Y 284.422,Z 509.868,A -85,B 0,C 180,E1 -16937.248,E2 -16937.248} C_VEL
LIN {X 0,Y 284.377,Z 509.873,A -85,B 0,C 180,E1 -16940.242,E2 -16940.242} C_VEL
LIN {X 0,Y 284.366,Z 509.876,A -85,B 0,C 180,E1 -16943.876,E2 -16943.876} C_VEL
LIN {X 0,Y 284.394,Z 509.872,A -85,B 0,C 180,E1 -16947.174,E2 -16947.174} C_VEL
LIN {X 0,Y 284.295,Z 509.885,A -85,B 0,C 180,E1 -16951.274,E2 -16951.274} C_VEL
LIN {X 0,Y 284.359,Z 509.877,A -85,B 0,C 180,E1 -16955.354,E2 -16955.354} C_VEL
LIN {X 0,Y 284.32,Z 509.879,A -85,B 0,C 180,E1 -16958.167,E2 -16958.167} C_VEL
LIN {X 0,Y 284.293,Z 509.883,A -85,B 0,C 180,E1 -16962.131,E2 -16962.131} C_VEL
LIN {X 0,Y 284.304,Z 509.881,A -85,B 0,C 180,E1 -16966.2,E2 -16966.2} C_VEL
LIN {X 0,Y 284.349,Z 509.876,A -85,B 0,C 180,E1 -16970.014,E2 -16970.014} C_VEL
LIN {X 0,Y 284.552,Z 510.049,A -85,B 0,C 180,E1 -16972.218,E2 -16972.218} C_VEL
LIN {X 0,Y 285.393,Z 514.846,A -85,B 0,C 180,E1 -16975.502,E2 -16975.502} C_VEL
LIN {X 0,Y 285.845,Z 518.754,A -85,B 0,C 180,E1 -16978.089,E2 -16978.089} C_VEL
LIN {X 0,Y 284.867,Z 524.993,A -85,B 0,C 180,E1 -16982.048,E2 -16982.048} C_VEL
LIN {X 0,Y 283.879,Z 532.368,A -85,B 0,C 180,E1 -16986.665,E2 -16986.665} C_VEL
LIN {X 0,Y 283.183,Z 539.302,A -85,B 0,C 180,E1 -16990.965,E2 -16990.965} C_VEL
LIN {X 0,Y 284.765,Z 552.479,A -85,B 0,C 180,E1 -16991.59,E2 -16991.59} C_VEL
LIN {X 0,Y 285.707,Z 562.204,A -85,B 0,C 180,E1 -16992.278,E2 -16992.278} C_VEL
LIN {X 0,Y 286.234,Z 570.585,A -85,B 0,C 180,E1 -16993.038,E2 -16993.038} C_VEL
LIN {X 0,Y 286.546,Z 578.949,A -85,B 0,C 180,E1 -16993.978,E2 -16993.978} C_VEL
LIN {X 0,Y 286.212,Z 585.716,A -85,B 0,C 180,E1 -16994.877,E2 -16994.877} C_VEL
LIN {X 0,Y 285.436,Z 592.431,A -85,B 0,C 180,E1 -16995.929,E2 -16995.929} C_VEL
LIN {X 0,Y 284.661,Z 598.975,A -85,B 0,C 180,E1 -16997.162,E2 -16997.162} C_VEL
LIN {X 0,Y 283.959,Z 605.181,A -85,B 0,C 180,E1 -16998.581,E2 -16998.581} C_VEL
LIN {X 0,Y 283.419,Z 610.322,A -85,B 0,C 180,E1 -17000.005,E2 -17000.005} C_VEL
LIN {X 0,Y 282.978,Z 614.582,A -85,B 0,C 180,E1 -17001.431,E2 -17001.431} C_VEL
LIN {X 0,Y 282.665,Z 618.094,A -85,B 0,C 180,E1 -17002.859,E2 -17002.859} C_VEL
LIN {X 0,Y 282.409,Z 622.135,A -85,B 0,C 180,E1 -17005.029,E2 -17005.029} C_VEL
LIN {X 0,Y 282.415,Z 624.815,A -85,B 0,C 180,E1 -17007.148,E2 -17007.148} C_VEL
LIN {X 0,Y 282.376,Z 625.866,A -85,B 0,C 180,E1 -17008.575,E2 -17008.575} C_VEL
LIN {X 0,Y 282.406,Z 626.422,A -85,B 0,C 180,E1 -17010.001,E2 -17010.001} C_VEL
LIN {X 0,Y 282.373,Z 626.493,A -85,B 0,C 180,E1 -17011.427,E2 -17011.427} C_VEL
LIN {X 0,Y 282.406,Z 626.078,A -85,B 0,C 180,E1 -17012.854,E2 -17012.854} C_VEL
LIN {X 0,Y 282.407,Z 625.086,A -85,B 0,C 180,E1 -17014.282,E2 -17014.282} C_VEL
LIN {X 0,Y 282.592,Z 622.631,A -85,B 0,C 180,E1 -17016.426,E2 -17016.426} C_VEL
LIN {X 0,Y 283.658,Z 617.798,A -85,B 0,C 180,E1 -17019.988,E2 -17019.988} C_VEL
LIN {X 0,Y 284.84,Z 613.849,A -85,B 0,C 180,E1 -17022.107,E2 -17022.107} C_VEL
LIN {X 0,Y 286.54,Z 608.623,A -85,B 0,C 180,E1 -17024.199,E2 -17024.199} C_VEL
LIN {X 0,Y 288.62,Z 602.011,A -85,B 0,C 180,E1 -17026.263,E2 -17026.263} C_VEL
LIN {X 0,Y 290.713,Z 595.199,A -85,B 0,C 180,E1 -17027.953,E2 -17027.953} C_VEL
LIN {X 0,Y 292.437,Z 588.739,A -85,B 0,C 180,E1 -17029.297,E2 -17029.297} C_VEL
LIN {X 0,Y 293.585,Z 581.451,A -85,B 0,C 180,E1 -17030.66,E2 -17030.66} C_VEL
LIN {X 0,Y 293.781,Z 573.368,A -85,B 0,C 180,E1 -17032.135,E2 -17032.135} C_VEL
LIN {X 0,Y 292.873,Z 563.577,A -85,B 0,C 180,E1 -17033.861,E2 -17033.861} C_VEL
